(* CODESYS project rsCommSerial.library
   Company: ESO
   Description: Library for Serial communication.
      Depends on rsCommCommon.library
   Version: 0.2.0.3
   Placeholder: ESO LDC Comm Serial Library
   Title: ESO LDC Comm Serial Library

Project tree, tasks and I/O mapping:
  libraries: ESO LDC Comm Common Library, 0.2.0.3 (ESO); Tc2_SerialCom, * (Beckhoff Automation GmbH); Tc2_Standard, * (Beckhoff Automation GmbH); Tc2_System, * (Beckhoff Automation GmbH); Tc2_Utilities, * (Beckhoff Automation GmbH); Tc3_Module, * (Beckhoff Automation GmbH); VisuDialogs, * (System)
  config/
    CCC__1HE_4HE__CoE.jpg
    EL6002_Lakeshore340.xti
    ic0fbiCCC_TwinCAT.fbmap
    LS218_CoE.jpg
    LS340_CoE.jpg
  00000000-0000-0000-0000-000000000000|config\CCC__1HE_4HE__CoE.jpg
  00000000-0000-0000-0000-000000000000|config\EL6002_Lakeshore340.xti
  00000000-0000-0000-0000-000000000000|config\ic0fbiCCC_TwinCAT.fbmap
  00000000-0000-0000-0000-000000000000|config\LS218_CoE.jpg
  00000000-0000-0000-0000-000000000000|config\LS340_CoE.jpg
  DUTs/
    Enumerated/
      Comm/
        data type E_MODBUS_CMD
        data type E_MODBUS_ERROR
        data type E_MODBUS_STATE
        data type E_MODBUS_STATUS
      Devices/
        data type E_CCC_ERROR
        data type E_CCC_STATUS
        data type E_JUMO_ADDRESS
    Structures/
      Comm/
        data type T_MODBUS_CFG
        data type T_MODBUS_CTRL
        data type T_MODBUS_INFO
        data type T_MODBUS_STAT
        data type T_USB_COMM_CFG
      Devices/
        data type T_CCC_CFG
        data type T_CCC_COMMAND
        data type T_CCC_CTRL
        data type T_CCC_INFO
        data type T_CCC_READING
        data type T_CCC_STAT
        data type T_JUMO_CFG
        data type T_JUMO_CTRL
        data type T_JUMO_INFO
        data type T_JUMO_STAT
  GVLs/
  lib/
  POUs/
    Comm/
      function block FB_MODBUS_COMM_BASE [ST]: M_ActionInitExecute, M_ActivityConnect, M_ComPortControl, M_CRC, M_GetHighByte, M_GetINT, M_GetLowByte, M_Reset
      function block FB_MODBUS_COMM_JUMO [ST]
      function block FB_MODBUS_COMM_NO_SIM [ST]
      function block FB_RS_COMM_BASE [ST]: M_ActionInitExecute, M_ActivityConnect, M_ComPortControl, M_GetInitialised, M_GetStatus, M_Reset
      function block FB_RS_COMM_LAKESHORE [ST]: M_ActionInitExecute, M_ComPortControl, M_Reset
      function block FB_RS_COMM_NO_SIM [ST]: M_ActionInitExecute, M_ComPortControl, M_Reset
      function block FB_USB_COMM_NO_SIM [ST]: M_ActionInitExecute, M_ActivityConnect, M_ComPortControl
    Devices/
      function block FB_CCC [ST]: ActivityInitializing, ActivityMonitoring, M_ConvertTemp, M_SetAllFaulty, M_TrimDevReply, M_UpdateDevFlows, M_UpdateDevStatus, M_UpdateDevTemps
      function block FB_JUMO [ST]: ActivityInitializing, ActivityMonitoring, M_ByteSwapFLOAT, M_ByteSwapINT, M_ExtractReadings, M_GetFirstSlaveIndex, M_GetNextSlaveIndex, M_SetCommand, M_UserConfigure
      function block FB_LAKESHORE_RS [ST]: M_Configure, M_GetCommInitialised, M_GetCommStatus, M_GetCouplerState, M_UpdateStatus
    program MAIN [ST]
  VISUs/
    Templates/
      visualisation GUI_TEMPLATE_CCC
      visualisation GUI_TEMPLATE_LAKESHORE_340
      visualisation GUI_TEMPLATE_USB_COMM
    visualisation GUI_ADS_COMM_TEST
    visualisation GUI_CCC
    visualisation GUI_LAKESHORE_340
  text list GlobalTextList
*)

// DUTs/Enumerated/Comm/E_MODBUS_CMD
{attribute 'qualified_only'}
////{xxxattribute 'strict'}
TYPE E_MODBUS_CMD :
(
	NONE		:=	0,
	INIT		:=	1,
	SEND		:=	2
);
END_TYPE

// DUTs/Enumerated/Comm/E_MODBUS_ERROR
{attribute 'qualified_only'}
//{xxxattribute 'strict'}
TYPE E_MODBUS_ERROR :
(
	OK					:= 0,
	NOT_IN_OP_STATE,
	NOT_INIT,
	TIMEOUT,
	SEND,
	RECEIVE,
	WRONG_STATE,
	NOT_IDLE
);
END_TYPE

// DUTs/Enumerated/Comm/E_MODBUS_STATE
{attribute 'qualified_only'}
{attribute 'strict'}
TYPE E_MODBUS_STATE :
(
	NOT_INIT			:= 0,
	IDLE				:= 1,
	RESET				:= 3,
	PREPARE_SEND		:= 5,
	SEND				:= 10,
	RECEIVE				:= 15,
	CLEAR_BUFFER		:= 40,

	ERROR				:= 100
);
END_TYPE

// DUTs/Enumerated/Comm/E_MODBUS_STATUS
{attribute 'qualified_only'}
////{xxxattribute 'strict'}
TYPE E_MODBUS_STATUS :
(
	NOT_INIT	:= -1,
	IDLE		:= 0,
	BUSY		:= 1,
	ERROR		:= 2
);
END_TYPE

// DUTs/Enumerated/Devices/E_CCC_ERROR
TYPE E_CCC_ERROR :
(
	OK				:= 16#0000,
	NOT_IN_OP_STATE	:= 16#0001,
	NOT_INIT		:= 16#0002,
	TIMEOUT			:= 16#0004,
	COMM			:= 16#0008,
	WRONG_STATE		:= 16#0010,
	NOT_IDLE		:= 16#0020
);
END_TYPE

// DUTs/Enumerated/Devices/E_CCC_STATUS
TYPE E_CCC_STATUS :
(
	NOT_INIT	:= -1,
	IDLE		:= 0,
	ERROR		:= 1,
	BUSY		:= 2
);
END_TYPE

// DUTs/Enumerated/Devices/E_JUMO_ADDRESS
TYPE E_JUMO_ADDRESS :
(
	COMMON		:=	0,
	SET_POINTS,
	END
);
END_TYPE

// DUTs/Structures/Comm/T_MODBUS_CFG
TYPE T_MODBUS_CFG EXTENDS T_RS_COMM_CFG:
STRUCT
END_STRUCT
END_TYPE

// DUTs/Structures/Comm/T_MODBUS_CTRL
TYPE T_MODBUS_CTRL :
STRUCT
	nCommand:	E_MODBUS_CMD 	:= E_MODBUS_CMD.NONE;			// Command Number, e.g. to INIT or SEND a command
	bExecute:	BOOL;								// Setting to TRUE activates command
	nSlaveID:	BYTE 	:= 1;						// Modbus Slave ID, 1..247
	nCmdType:	E_MODBUS_CMD_TYPE	:= E_MODBUS_CMD_TYPE.READ;	// Command type; 0-Read, 1-Write
	nRegister:	DINT;								// Command register
	nWords:		DINT	:= 1;						// Number of words
	nValue:		DINT;								// Parameter value

END_STRUCT
END_TYPE

// DUTs/Structures/Comm/T_MODBUS_INFO
TYPE T_MODBUS_INFO :
STRUCT
(*
	Driver Information

	Change LOG:
	01/09/2016:	0.1	- First version. Based on FB_RS_COMM.
	05/09/2016:	0.2	- Implemented Modbus protocol.
	09/11/2016:	0.3	- Status cleared on INIT.
*)

	sDate:			STRING(32)	:= '2016-11-09';
	sDescription:	STRING(80) 	:= 'IR-301 Black Body RS-232 Modbus Driver';
	sName:			STRING(64)	:= 'FB_RS_COMM';
	sPlatform:		STRING(32)	:= 'CoDeSys';
	sSynopsis:		STRING(64)	:= 'IR-301 Black Body RS-232 Modbus Driver';
	nVersionMajor:	DINT		:= 0;
	nVersionMinor:	DINT		:= 3;


END_STRUCT
END_TYPE

// DUTs/Structures/Comm/T_MODBUS_STAT
TYPE T_MODBUS_STAT EXTENDS T_RS_COMM_STAT:
STRUCT
	DeviceReply: 		ARRAY [0..300] OF BYTE;
	nValue:				DINT;	// Value read from the device
END_STRUCT
END_TYPE

// DUTs/Structures/Comm/T_USB_COMM_CFG
TYPE T_USB_COMM_CFG EXTENDS T_RS_COMM_CFG:
STRUCT
	ComPort: 		UDINT :=5;         					// Serial port number [1..255]
    Baudrate: 		UDINT :=57600;						// Baudrate
    Parity: 		ComParity_t :=ComParity_t.PARITY_NONE;			// PARITY_NONE, _EVEN, _ODD, _MARK or _SPACE
    DataBits: 		INT :=8;           					// Data Bits [4..8]
    StopBits: 		ComStopBits_t :=ComStopBits_t.STOPBITS_ONE;		// Stop Bits

    DTR: 			ComDTRCtrl_t :=ComDTRCtrl_t.DTR_CTRL_DISABLE; 	// DTR_CTRL_DISABLE, _ENABLE or _HANDSHAKE
    RTS: 			ComRTSCtrl_t :=ComRTSCtrl_t.RTS_CTRL_DISABLE; 	// RTS_CTRL_DISABLE, _ENABLE, _HANDSHAKE or _TOGGLE
    CTS: 			BOOL :=FALSE;      					// 'Clear to Send' signal
    DSR: 			BOOL :=FALSE;      					// 'Dataset Ready' signal

END_STRUCT
END_TYPE

// DUTs/Structures/Devices/T_CCC_CFG
TYPE T_CCC_CFG EXTENDS T_RS_BASE_CFG:
STRUCT
	CCC_CMD_GET_VERS:	STRING(8) := '>00V??';
	CCC_CMD_RESET:		STRING(8) := '>00u??';
	CCC_CMD_GET_TEMP:	STRING(8) := '>00H??';
	CCC_CMD_GET_FLOW:	STRING(8) := '>00f??';
	CCC_CMD_GET_STAT:	STRING(8) := '>00o??';
	CCC_CMD_SET_HOST:	STRING(8) := '>00J??';
	CCC_CMD_SET_THST:	STRING(8) := '>00T??';
	CCC_CMD_SET_TAMB:	STRING(8) := '>00t??';

	(* List of INIT commands *)
	cmdList_Init:	ARRAY [1..4] OF T_CCC_COMMAND := [
							(cmd := CCC_CMD_RESET, 		nValues := 0),
							(cmd := CCC_CMD_GET_VERS, 	nValues := 0),
							(cmd := '', 				nValues := 0),
							(cmd := '', 				nValues := 0)];


	(*	List of READ commands *)
	cmdList_Read:	ARRAY [1..4] OF T_CCC_COMMAND := [
							(cmd := CCC_CMD_GET_STAT, 	nValues := 5), (* 5 bytes *)
							(cmd := CCC_CMD_GET_TEMP, 	nValues := 5), (* 5 words = 10 bytes*)
							(cmd := CCC_CMD_GET_FLOW, 	nValues := 3), (* 3 words = 6 bytes *)
							(cmd := '', 				nValues := 0)];

END_STRUCT
END_TYPE

// DUTs/Structures/Devices/T_CCC_COMMAND
TYPE T_CCC_COMMAND :
STRUCT
	cmd:		STRING(8);	(* Command to send *)
	nValues:	DINT;   	(* Number of returned numbers (values) in the reply *)
END_STRUCT
END_TYPE

// DUTs/Structures/Devices/T_CCC_CTRL
TYPE T_CCC_CTRL  EXTENDS T_RS_BASE_CTRL:
STRUCT
	(* CTRL *)
END_STRUCT
END_TYPE

// DUTs/Structures/Devices/T_CCC_INFO
TYPE T_CCC_INFO :
STRUCT
(*
	Driver Information

	Change LOG:
	1.0	12/02/2014	- Ported from TC2.
	1.1	13/02/2014	- Addition of input parameters for Model and readout period.
	1.2	20/02/2014	- E_CCC_STATUS.ERROR := 1, to match IODev ICD.
					- Disabled OPC UA for comm instance of FB_RS_COMM.
					- Fixed bug in INIT (wrong pointer used)
					- Bytes swapped for Temperatures and Flows.
					- On error, all values set to 9999. Alarm activated.
	1.3 07/11/2014	- Newest version always for References.
					- Remove Tc2_OpcUa library from References.
					- Renamed library to CCC.library (was CCC_TC3.library)
					- Created lib directory.
	1.4 10/02/2016	- On reboot, the device is in NOT INIT (no error!)
					- On INIT start, error is cleared.
	2.0 2016-08-10	- OPC UA notation with TMC Files
	2.1 2017-02-03	- sCmdSuffix and sReplySuffix passed to comm instance.

*)
	sDate:			STRING(16)	:= '2017-02-03';
	sDescription:	STRING(32) 	:= 'Cabinet Cooling Controller';
	sName:			STRING(16)	:= 'FB_CCC';
	sPlatform:		STRING(16)	:= 'CoDeSys';
	sSynopsis:		STRING(48)	:= 'Cabinet Cooling Controller for models 1HE & 4HE';
	nVersionMajor:	DINT		:= 2;
	nVersionMinor:	DINT		:= 1;

END_STRUCT
END_TYPE

// DUTs/Structures/Devices/T_CCC_READING
TYPE T_CCC_READING :
STRUCT
	Value:	LREAL;
END_STRUCT
END_TYPE

// DUTs/Structures/Devices/T_CCC_STAT
TYPE T_CCC_STAT EXTENDS T_RS_BASE_STAT:
STRUCT
	(* STAT *)
	nRetries:			INT := 0;			// Total number of retries in case of communication problems
	
	bPeriodic:			BOOL := FALSE;		(* Flag if device is reading periodically *)

	sReply:				STRING; 			(* Last Reply to predefined commands*)
	
	sDeviceID:			STRING(48);
	
	(* Status retrieved with command CCC_CMD_GET_STAT *)
	(* decode CSTAT1 byte *)
	bWarn_cabinet_high:			BOOL;
	bWarn_cabinet_no_control:	BOOL;
	bWarn_outlet_high:			BOOL;
	bWarn_inlet_high:			BOOL;
	bWarn_airflow_insufficient:	BOOL;
	bWarn_coolant_insufficient:	BOOL;
	bWarn_door_open:			BOOL;
	bWarn_relay1_warning:		BOOL;
	bWarn_relay2_alarm:			BOOL;

	(* decode CSTAT2 byte *)
	bFault_temp_sensor_ambient:	BOOL;
	bFault_temp_sensor_cabinet:	BOOL;
	bFault_temp_sensor_inlet:	BOOL;
	bFault_temp_sensor_outlet:	BOOL;
	bFault_analog_supply:		BOOL;
	bFault_digital_supply:		BOOL;
	
	(* Temperatures [degC] retrieved with command CCC_CMD_GET_TEMP *)
	lrTemp_outlet:	LREAL;
	lrTemp_inlet:	LREAL;
	lrTemp_cabinet:	LREAL;
	lrTemp_ambient:	LREAL;
	
	(* Flows [l/h] retrieved with command CCC_CMD_GET_FLOW *)
	lrFlow_1:		LREAL;
	lrFlow_2:		LREAL;
	lrFlow_3:		LREAL;

END_STRUCT
END_TYPE

// DUTs/Structures/Devices/T_JUMO_CFG
TYPE T_JUMO_CFG EXTENDS T_RS_BASE_CFG:
STRUCT
	// Register Addresses
	nAddrCommon:		INT	:= 16#00A4;
	nAddrSetPoints:		INT	:= 16#083C;

	// Number of bytes to read
	// These are ONLY data bytes. Total bytes to read is higher (+5) 
	nWordsCommon:		INT	:= 116;	// 232 bytes
	nWordsSetPoints:	INT	:= 32;	// 32 words
	
	aSlaveID:			ARRAY [1..8] OF BYTE := [1,2,3,4,5,6,7,8];
	aDevUsed:			ARRAY [1..8] OF BOOL := [TRUE, 7(FALSE)];	// Only first JUMO used by default
	
END_STRUCT
END_TYPE

// DUTs/Structures/Devices/T_JUMO_CTRL
TYPE T_JUMO_CTRL EXTENDS T_RS_BASE_CTRL:
STRUCT
	nSlaveID:	BYTE 	:= 1;						// Modbus Slave ID, 1..247
	nCmdType:	DINT	:= E_MODBUS_CMD_TYPE.READ;	// Command type; 0-Read, 1-Write
	nRegister:	DINT;								// Command register
	nWords:		DINT	:= 1;						// Number of words
	nValue:		DINT;								// Parameter value
END_STRUCT
END_TYPE

// DUTs/Structures/Devices/T_JUMO_INFO
TYPE T_JUMO_INFO :
STRUCT
(*
	Driver Information

	Change LOG:
	1.0	12/02/2014	- Copied from VLT.
*)
	sDate:			STRING(16)	:= '2016-08-10';
	sDescription:	STRING(32) 	:= 'JUMO controller';
	sName:			STRING(16)	:= 'FB_JUMO';
	sPlatform:		STRING(16)	:= 'CoDeSys';
	sSynopsis:		STRING(48)	:= 'EtherCAT PLC JUMO controller';
	nVersionMajor:	DINT		:= 1;
	nVersionMinor:	DINT		:= 0;

END_STRUCT
END_TYPE

// DUTs/Structures/Devices/T_JUMO_STAT
TYPE T_JUMO_STAT EXTENDS T_RS_BASE_STAT:
STRUCT

	nRetries:				INT := 0;	// Total number of retries in case of communication problems
	
	nInputBuffer: 			ARRAY [0..300] OF BYTE;	// Binary data read from JUMO

	// Data for up to 8 JUMO devices (4 TeePee units) daisy chained
	// Data for the first 4 control loops [1-4]
	// ARRAY[<device>,<control loop>, <value>]
	aSetPoints:				ARRAY [1..8,1..4,1..4] OF REAL;
	aCtrlParams:			ARRAY [1..8,1..4,1..9] OF REAL;
	aSwitchStats:			ARRAY [1..8,1..4,1..2] OF INT;

	// 8 analog inputs per JUMO
	aAnalogInputs:			ARRAY [1..8,1..8] OF REAL;
	aMath:					ARRAY [1..8,1..8] OF REAL;

	aSamplingTime:			ARRAY [1..8] OF REAL;
	aInternalTemperature:	ARRAY [1..8] OF REAL;
END_STRUCT
END_TYPE

// POUs/Comm/FB_MODBUS_COMM_BASE
FUNCTION_BLOCK FB_MODBUS_COMM_BASE
VAR_INPUT
	in_bSimulation:		BOOL := FALSE;
	in_nModel:			DINT;	// Device model number. Zero if N/A.
	in_cReadFunction:	BYTE := 3;	// Function used for READ. MUST be 3 or 4.
END_VAR
VAR_OUTPUT
END_VAR
VAR CONSTANT
END_VAR
VAR
	{attribute 'OPC.UA.DA' := '1'}
	cfg:		T_MODBUS_CFG;				// Config parameters
	{attribute 'OPC.UA.DA' := '1'}
	ctrl:		T_MODBUS_CTRL;				// Control parameters
	{attribute 'OPC.UA.DA' := '1'}
	{attribute 'OPC.UA.DA.Access' := '1'}
	info:		T_MODBUS_INFO; 				// Info parameters - ReadOnly
	{attribute 'OPC.UA.DA' := '1'}
	{attribute 'OPC.UA.DA.Access' := '1'}
	stat:		T_MODBUS_STAT;				// Status parameters - ReadOnly

	{attribute 'OPC.UA.DA' := '0'}
	simRef:		REFERENCE TO FB_SIM_MODBUS_COMM_BASE;	// Reference to COMM simulator


	(***** Physical signals - to be mapped to EL60xx serial port terminal !!! *****)
	COMin_EL60xx	AT %I* 	: KL6inData22B;	(* linked to the EL60xx *)
	COMout_EL60xx	AT %Q*	: KL6outData22B;(* linked to the EL60xx *)
	i_nCouplerState	AT %I*	: UINT;			(* Link it to Coupler->InfoData->State *)

	(* Serial line control *)
	COMportControl: 		SerialLineControl;
	RxBuffer:				ComBuffer;		(* Receive data buffer; used with all receive function blocks *)
	TxBuffer:				ComBuffer;		(* Transmit data buffer; used with all receive function blocks *)


	(* Send/Receive FB's and VAR's *)
	Receive: 			ReceiveData;
	Send:				SendData;
	ClearComBufferTx:	ClearComBuffer;
	ClearComBufferRx:	ClearComBuffer;
	ComReset:			ComReset;

	(* Timers *)
	fbTimer:			TON; (* Timeout for RECEIVE *)

	State:				INT := E_MODBUS_STATE.NOT_INIT;
	nextState:			INT := E_MODBUS_STATE.IDLE;


	cmd:				STRING(16);		// Only first 8 bytes are used

	nBytesToReceive:	UDINT;			// 8 for command, 7 for status
	nBytesToSend:		UDINT := 8;		// Always 8

	crc:				WORD;			// CRC Check word

	i:					INT;
END_VAR

(* ============================================
	Check if the HW is OK. 
	The coupler state must be 8, i.e. OPERATIONAL.
============================================== *)
IF i_nCouplerState <> 8  AND  NOT in_bSimulation THEN	(* If the hardware status is NOT OK, we cannot trust the readings. *)
	stat.nErrorCode	:= M_GetINT(E_MODBUS_ERROR.NOT_IN_OP_STATE);
	stat.sErrorText	:= 'Not in OPERATIONAL state. Check if variable i_nCouplerState is linked to HW.';
	stat.nStatus	:= M_GetINT(E_MODBUS_STATUS.ERROR);
	stat.sStatus	:= 'ERROR';
	RETURN;
END_IF


//
// Execute Simulator, if in simulation
//
IF in_bSimulation  THEN
	simRef(in_nModel := in_nModel);
END_IF


(*====================================================
	Handling of commands sent through OPC UA interface.
	Executed only when flag bExecute goes from LOW to HIGH.
	bExecute is reset by the PLC application.
=====================================================*)

IF ctrl.bExecute THEN
	ctrl.bExecute	:= FALSE;
	(* Save last command and reset the command *)
	stat.nLastCommand 	:= M_GetINT(ctrl.nCommand);
	ctrl.nCommand		:= E_MODBUS_CMD.NONE;

	(* Commands can only be sent when device is IDLE *)
	IF INT_TO_DINT(stat.nLastCommand) <> INT_TO_DINT(E_MODBUS_CMD.INIT)  AND  State <> E_MODBUS_STATE.IDLE THEN
		State 			:= E_MODBUS_STATE.ERROR;
		stat.nStatus	:= M_GetINT(E_MODBUS_STATUS.ERROR);
		stat.sStatus	:= 'ERROR';
		stat.nErrorCode	:= M_GetINT(E_MODBUS_ERROR.NOT_IDLE);
		stat.sErrorText	:= 'Device busy. Should be in IDLE to receive commands.';
		RETURN;
	END_IF


	(* Device has to be initialised before being used *)
	IF INT_TO_DINT(stat.nLastCommand) <> INT_TO_DINT(E_MODBUS_CMD.INIT) THEN
		IF NOT stat.bInitialised  THEN
			State 			:= E_MODBUS_STATE.ERROR;
			stat.nStatus	:= M_GetINT(E_MODBUS_STATUS.ERROR);
			stat.sStatus	:= 'ERROR';
			stat.nErrorCode	:= M_GetINT(E_MODBUS_ERROR.NOT_INIT);
			stat.sErrorText	:= 'Device not initialised.';
			RETURN;
		END_IF
	END_IF



	CASE stat.nLastCommand OF
	E_RS_COMM_CMD.INIT:
		// Comm port specific.
		// M_ActionInitExecute() has to set next State!!!
		M_ActionInitExecute();

	E_RS_COMM_CMD.SEND:
		stat.nErrorCode	:= M_GetINT(E_MODBUS_ERROR.OK);
		stat.nStatus	:= M_GetINT(E_MODBUS_STATUS.BUSY);
		stat.sErrorText	:= 'OK';
		stat.sStatus	:= 'BUSY';
		State 			:= E_MODBUS_STATE.PREPARE_SEND;

	END_CASE

END_IF



(*====================================================
	Background communication with KL60xx terminal.
	Called only during Send or Receive!!!
	It communicates with the serial line hardware device and 
	transmits or receives data.
=====================================================*)

CASE State OF
E_MODBUS_STATE.IDLE,
E_MODBUS_STATE.CLEAR_BUFFER,
E_MODBUS_STATE.SEND,
E_MODBUS_STATE.RECEIVE:

	COMportControl(
		Mode		:= ComSerialLineMode_t.SERIALLINEMODE_KL6_22B_STANDARD,
		pComIn		:= ADR(COMin_EL60xx),				(* I/O data; see global variables *)
		pComOut		:= ADR(COMout_EL60xx),				(* I/O data; see global variables *)
		SizeComIn	:= UINT_TO_INT(SIZEOF(COMin_EL60xx)),			(* I/O data; see global variables *)
		TxBuffer	:= TxBuffer,						(* transmit buffer; see global variables *)
		RxBuffer	:= RxBuffer);						(* receive buffer; see global variables *)

END_CASE





(*======================
=======================
 	State machine 
=======================
=======================*)

CASE State OF

E_MODBUS_STATE.ERROR:
	ClearComBufferTx (Buffer := TxBuffer);
	ClearComBufferRx (Buffer := RxBuffer);
	stat.nStatus	:= M_GetINT(E_MODBUS_STATUS.ERROR);
	stat.sStatus	:= 'ERROR';
	State 			:= E_MODBUS_STATE.IDLE;
	RETURN;


E_MODBUS_STATE.NOT_INIT:
	ClearComBufferTx (Buffer := TxBuffer);
	ClearComBufferRx (Buffer := RxBuffer);
	stat.bInitialised	:= FALSE;
	stat.nErrorCode		:= M_GetINT(E_MODBUS_ERROR.OK);
	stat.sErrorText		:= 'OK';
	stat.nStatus		:= M_GetINT(E_MODBUS_STATUS.NOT_INIT);
	stat.sStatus		:= 'NOT INIT';


E_MODBUS_STATE.IDLE:
	(* Nothing to do in IDLE *)
	RETURN;


E_MODBUS_STATE.RESET:
	(* Reset the connected serial hardware *)
	ComReset (
		Execute 	:= TRUE,
		pComIn		:= ADR(COMin_EL60xx),
		pComOut		:= ADR(COMout_EL60xx),
		SizeComIn	:= SIZEOF(COMin_EL60xx),
		);

	(* Next step is to clear the buffers *)
	IF ComReset.Done THEN
		fbTimer (IN := FALSE);	// Reset the timer
		State 		:= E_MODBUS_STATE.CLEAR_BUFFER;
	END_IF
	RETURN;


E_MODBUS_STATE.PREPARE_SEND:
	(*******************************************************************************************
	Here we set the command string, i.e. add suffix if not included in the command.
	Then, the state is changed to  E_MODBUS_STATE.SEND.
	********************************************************************************************)

	(* Clear reply string *)
	MEMSET(ADR(stat.DeviceReply), 0 , SIZEOF(stat.DeviceReply) );

	cmd	:= '';
	cmd[0] := ctrl.nSlaveID;
	cmd[2] := M_GetHighByte(ctrl.nRegister);
	cmd[3] := M_GetLowByte(ctrl.nRegister);
	IF ctrl.nCmdType = E_MODBUS_CMD_TYPE.WRITE  THEN
		cmd[1] := 6;			// Write Function
		nBytesToReceive	:= 8;	// Reply equals Command
		cmd[4] := M_GetHighByte(ctrl.nValue);
		cmd[5] := M_GetLowByte(ctrl.nValue);
	ELSE
		cmd[1] := in_cReadFunction;			// Read Function (3 or 4)
		nBytesToReceive	:= DINT_TO_UDINT(2 * ctrl.nWords  +  5); 
		// Bytes 4..5, receive one word (2 bytes)
		cmd[4] := M_GetHighByte(ctrl.nWords);
		cmd[5] := M_GetLowByte(ctrl.nWords);
	END_IF
	
	// Calculate CRC for the first 6 bytes
	crc	:= M_CRC(ADR(cmd),6);
	
	cmd[6] := M_GetLowByte(crc);
	cmd[7] := M_GetHighByte(crc);
	
	IF in_bSimulation THEN
		fbTimer (IN := FALSE); 	(* reset timer *)
		ClearComBufferRx (Buffer := RxBuffer);
		stat.sReply		:= simRef.M_GetSimReply(cmd);	// Get simulated reply
		FOR i:=0 TO 255 DO
			stat.DeviceReply[i] := stat.sReply[i];
		END_FOR
		stat.nStatus	:= M_GetINT(E_MODBUS_STATUS.IDLE);
		stat.sStatus	:= 'IDLE';
		State 			:= E_MODBUS_STATE.IDLE;
	ELSE	
		ClearComBufferTx (Buffer := TxBuffer);
		stat.nStatus	:= M_GetINT(E_MODBUS_STATUS.BUSY);
		stat.sStatus	:= 'BUSY';
		State 			:= E_MODBUS_STATE.SEND;
	END_IF
	RETURN;


E_MODBUS_STATE.SEND:

	(* Send the command via serial port. *)
	Send(
		pSendData	:= ADR(cmd),
		Length		:= nBytesToSend,
		TXbuffer	:= TxBuffer);

	(* If the string was not sent in one cycle, go to next cycle *)
	IF Send.Busy THEN
		RETURN;
	ELSE
		IF Send.Error <> ComError_t.COMERROR_NOERROR THEN
			State 			:= E_MODBUS_STATE.ERROR;
			stat.nErrorCode	:= M_GetINT(E_MODBUS_ERROR.SEND);
			stat.sErrorText	:= 'Send Failed';
		ELSE
			fbTimer (IN := FALSE);	// reset timer
			// One extra call of background communication
			COMportControl(
				Mode		:= ComSerialLineMode_t.SERIALLINEMODE_KL6_22B_STANDARD,
				pComIn		:= ADR(COMin_EL60xx),				(* I/O data; see global variables *)
				pComOut		:= ADR(COMout_EL60xx),				(* I/O data; see global variables *)
				SizeComIn	:= UINT_TO_INT(SIZEOF(COMin_EL60xx)),			(* I/O data; see global variables *)
				TxBuffer	:= TxBuffer,						(* transmit buffer; see global variables *)
				RxBuffer	:= RxBuffer);						(* receive buffer; see global variables *)

			State := E_MODBUS_STATE.RECEIVE; 	(* Next state is RECEIVE *)
		END_IF
		RETURN;
	END_IF



E_MODBUS_STATE.RECEIVE:
	(* Start the 3 sec timeout timer for receive *)
	fbTimer (IN := TRUE, PT := T#3S);

	(* Check for timeout. Goto ERROR if timeout expired. *)
	IF fbTimer.Q THEN
		fbTimer (IN := FALSE); (* reset timer *)

		State 			:= E_MODBUS_STATE.ERROR;
		stat.nErrorCode	:= M_GetINT(E_MODBUS_ERROR.TIMEOUT);
		stat.sErrorText	:= 'Timeout on Receive';
		RETURN;
	END_IF

	// Wait for the reply.
	// Terminate read 1000 ms after receiving the first character.
	Receive(
		pReceiveData	:= ADR(stat.DeviceReply),
		SizeReceiveData := nBytesToReceive,
		Timeout			:= T#1000MS,
		Reset			:= FALSE,
		RXbuffer		:= RxBuffer);


	(* Check for possible errors *)
	IF Receive.Error <> ComError_t.COMERROR_NOERROR THEN
		fbTimer (IN := FALSE);	(* reset timer *)

		State 			:= E_MODBUS_STATE.ERROR;
		stat.nErrorCode	:= M_GetINT(E_MODBUS_ERROR.RECEIVE);
		stat.sErrorText	:= 'Receive Failed';
		RETURN;
	END_IF

	(* Handle reply *)
	IF Receive.DataReceived THEN
		(* We have received a reply. Reset timers and triggers. *)
		fbTimer (IN := FALSE); 	(* reset timer *)

		// Calculate CRC for the first (nBytesToReceive-2) bytes.
		// The last two bytes are the CRC returned by the device.
		// Do a CRC check.
		crc	:= M_CRC(ADR(stat.DeviceReply),UDINT_TO_INT(nBytesToReceive-2));
		
		IF stat.DeviceReply[nBytesToReceive-1] <> M_GetHighByte(crc) THEN
			State 			:= E_MODBUS_STATE.ERROR;
			stat.nErrorCode	:= M_GetINT(E_MODBUS_ERROR.RECEIVE);
			stat.sErrorText	:= 'Received CRC does not match';
			RETURN;
		ELSIF stat.DeviceReply[nBytesToReceive-2] <> M_GetLowByte(crc) THEN
			State 			:= E_MODBUS_STATE.ERROR;
			stat.nErrorCode	:= M_GetINT(E_MODBUS_ERROR.RECEIVE);
			stat.sErrorText	:= 'Received CRC does not match';
			RETURN;
		END_IF
	
		
		(* Clear the receive buffer ONLY when all replies have been received! *)
		ClearComBufferRx (Buffer := RxBuffer);
		State 			:= E_MODBUS_STATE.IDLE;
		stat.nStatus	:= M_GetINT(E_MODBUS_STATUS.IDLE);
		stat.sStatus	:= 'IDLE';
		RETURN;
	ELSIF Receive.RxTimeout THEN
		(* Handle reply *)
		(* We have received a reply. Reset timers and triggers. *)
		fbTimer (IN := FALSE); 	(* reset timer *)

		// Clear the receive buffer
		ClearComBufferRx (Buffer := RxBuffer);

		stat.nErrorCode	:= M_GetINT(E_MODBUS_ERROR.TIMEOUT);
		stat.sErrorText	:= 'Did not receive expected number of bytes';

		State 			:= E_MODBUS_STATE.ERROR;
		RETURN;
	END_IF



E_MODBUS_STATE.CLEAR_BUFFER:
	// Read all characters present in the receive buffer.
	// Keep reading for 1 sec.
	fbTimer (IN := TRUE, PT := T#1S);
	IF fbTimer.Q THEN
		(* reset timer *)
		fbTimer (IN := FALSE);
		stat.bInitialised	:= TRUE;
		stat.nStatus		:= M_GetINT(E_MODBUS_STATUS.IDLE);
		stat.sStatus		:= 'INITIALISED';
		State 				:= E_MODBUS_STATE.IDLE;
		RETURN;
	END_IF

	Receive(
		pReceiveData	:= ADR(stat.DeviceReply),
		SizeReceiveData := SIZEOF(nBytesToReceive),
		Timeout			:= T#300MS,
		Reset			:= FALSE,
		RXbuffer		:= RxBuffer);



ELSE
(* Unsuported state *)
	State 			:= E_MODBUS_STATE.ERROR;
	stat.nErrorCode	:= M_GetINT(E_MODBUS_ERROR.WRONG_STATE);
	stat.sErrorText	:= 'Unknown State';
END_CASE

METHOD M_ActionInitExecute
VAR_INPUT
END_VAR
//
// If in simulation, there is no need to reset anything.
// Just set it to initialised and go to IDLE state.
//
IF in_bSimulation THEN
	fbTimer (IN := FALSE);	// Reset timer
	stat.bInitialised	:= TRUE;
	stat.nStatus		:= M_GetINT(E_MODBUS_STATUS.IDLE);
	stat.sStatus		:= 'INITIALISED';
	State 				:= E_MODBUS_STATE.IDLE;
ELSE
	stat.bInitialised	:= FALSE;
	stat.sStatus		:= 'INITIALISING';
	stat.nStatus		:= M_GetINT(E_MODBUS_STATUS.BUSY);
	stat.nErrorCode		:= M_GetINT(E_MODBUS_ERROR.OK);
	stat.sErrorText		:= 'OK';

	// Reset the connected serial hardware 
	ComReset (
		Execute 	:= FALSE,
		pComIn		:= ADR(COMin_EL60xx),
		pComOut		:= ADR(COMout_EL60xx),
		SizeComIn	:= SIZEOF(COMin_EL60xx),
		);

	// Set next state
	State 	:= E_MODBUS_STATE.RESET;
END_IF
END_METHOD

METHOD M_ActivityConnect
VAR_INPUT
END_VAR
// TODO: Implement in extended FB
END_METHOD

METHOD M_ComPortControl
VAR_INPUT
END_VAR
// TODO: Implement in extended FB
END_METHOD

METHOD M_CRC : WORD
VAR_INPUT
	p:	POINTER TO BYTE;
	n:	INT;
END_VAR
VAR
  crc: 			WORD;
  bit_count: 	BYTE;
  char_ptr: 	POINTER TO BYTE;
  pos:			INT := 0;
END_VAR
VAR CONSTANT
	POLYNOMIAL: WORD := 16#A001;
END_VAR

// Start at the beginning of the packet
char_ptr := p;

// Initialize CRC
crc := 16#FFFF;

// Loop through the entire packet
WHILE pos < n DO
	
	  // Exclusive-OR the byte with the CRC
	crc := crc XOR char_ptr^;		// crc ^= (unsigned int)*char_ptr;
	
	  // Loop through all 8 data bits
	  bit_count := 0;
	  WHILE bit_count < 8 DO
		  // If the LSB is 1, shift the CRC and XOR
		  // the polynomial mask with the CRC
		  IF (crc AND 16#0001) <> 16#0000 THEN
			
			  crc := SHR(crc,1);	// crc >>= 1;
			  crc := crc XOR POLYNOMIAL;	// crc ^= POLYNOMIAL;
			
		  // If the LSB is 0, shift the CRC only
		  else
			crc := SHR(crc,1);	// crc >>= 1;			
		END_IF
		bit_count := bit_count + 1;
	  END_WHILE
	  char_ptr := char_ptr + 1;
	  pos := pos + 1;
END_WHILE

M_CRC := crc;
END_METHOD

METHOD M_GetHighByte : BYTE
VAR_INPUT
	n:	DINT;
END_VAR
VAR
	w:	WORD;
END_VAR
w := DINT_TO_WORD(n);
M_GetHighByte	:= WORD_TO_BYTE(SHR((w AND 16#FF00), 8));
END_METHOD

METHOD M_GetINT : INT
VAR_INPUT
	nInt:	INT;
END_VAR
M_GetINT	:= nInt;
END_METHOD

METHOD M_GetLowByte : BYTE
VAR_INPUT
	n:	DINT;
END_VAR
VAR
	w:	WORD;
END_VAR
w := DINT_TO_WORD(n);
M_GetLowByte	:= WORD_TO_BYTE((w AND 16#00FF));
END_METHOD

METHOD M_Reset
VAR_INPUT
END_VAR
// TODO: Implement in extended FB
END_METHOD

END_FUNCTION_BLOCK

// POUs/Comm/FB_MODBUS_COMM_JUMO
FUNCTION_BLOCK FB_MODBUS_COMM_JUMO EXTENDS FB_MODBUS_COMM_BASE
VAR_INPUT
END_VAR
VAR_OUTPUT
END_VAR
VAR CONSTANT
END_VAR
VAR
	{attribute 'OPC.UA.DA' := '0'}
	sim:		FB_SIM_MODBUS_COMM_JUMO;	// Reference to COMM simulator

END_VAR

simRef	REF=sim;

// Execute base FB, i.e. FB_MODBUS_COMM_BASE.
SUPER^();

END_FUNCTION_BLOCK

// POUs/Comm/FB_MODBUS_COMM_NO_SIM
FUNCTION_BLOCK FB_MODBUS_COMM_NO_SIM EXTENDS FB_MODBUS_COMM_BASE
VAR_INPUT
END_VAR
VAR_OUTPUT
END_VAR
VAR CONSTANT
END_VAR
VAR
	{attribute 'OPC.UA.DA' := '0'}
	sim:		FB_SIM_MODBUS_COMM_BASE;	// Reference to COMM simulator

END_VAR

simRef	REF=sim;

// Execute base FB, i.e. FB_MODBUS_COMM_BASE.
SUPER^();

END_FUNCTION_BLOCK

// POUs/Comm/FB_RS_COMM_BASE
FUNCTION_BLOCK FB_RS_COMM_BASE
VAR_INPUT
	in_bSimulation:		BOOL := FALSE;
	in_nModel:			DINT;	// Device model number. Zero if N/A.
	in_sCmdSuffix:		STRING(16) := '$0D$0A';	// Terminator for command, default '<CR><LF>'
	in_sReplySuffix:	STRING(16) := '$0D$0A';	// Terminator for reply, default '<CR><LF>'
	in_nTimeout:		DINT := 3000;			// Timeout [ms] on command reply. Default 3000 (3 sec)
END_VAR
VAR_OUTPUT
END_VAR
VAR CONSTANT
END_VAR
VAR
	{attribute 'OPC.UA.DA' := '1'}
	cfgRef:			REFERENCE TO T_RS_COMM_CFG;		// Config parameters
	{attribute 'OPC.UA.DA' := '1'}
	ctrlRef:		REFERENCE TO T_RS_COMM_CTRL;	// Control parameters
	{attribute 'OPC.UA.DA' := '1'}
	{attribute 'OPC.UA.DA.Access' := '1'}
	infoRef:		REFERENCE TO T_RS_COMM_INFO; 	// Info parameters - ReadOnly
	{attribute 'OPC.UA.DA' := '1'}
	{attribute 'OPC.UA.DA.Access' := '1'}
	statRef:		REFERENCE TO T_RS_COMM_STAT;	// Status parameters - ReadOnly

	{attribute 'OPC.UA.DA' := '0'}
	simRef:			REFERENCE TO FB_SIM_RS_COMM_BASE;	// Reference to COMM simulator


	// Physical signals - to be mapped
	i_nCouplerState	AT %I*	: UINT;			(* Link it to Coupler->InfoData->State *)

	(* Serial line control *)
//	COMportControl: 		SerialLineControl;
	RxBuffer:				ComBuffer;		(* Receive data buffer; used with all receive function blocks *)
	TxBuffer:				ComBuffer;		(* Transmit data buffer; used with all receive function blocks *)

	(* Send/Receive FB's and VAR's *)
	Receive: 			ReceiveString255;
	Send:				SendString;
	ClearComBufferTx:	ClearComBuffer;
	ClearComBufferRx:	ClearComBuffer;
	ComReset:			ComReset;

	DeviceReply: 		STRING(255);

	(* Timers *)
	fbTimer:			TON; (* Timeout for RECEIVE *)

	State:				INT := E_RS_COMM_STATE.NOT_INIT;
	nextState:			INT := E_RS_COMM_STATE.IDLE;

	cmd:				STRING;

	nNumReplies:		DINT := 0;

	pos:				INT;
END_VAR

(* ============================================
	Check if the HW is OK. 
	The coupler state must be 8, i.e. OPERATIONAL (if not simulated).
============================================== *)
IF i_nCouplerState <> 8  AND  NOT in_bSimulation  THEN	(* If the hardware status is NOT OK, we cannot trust the readings. *)
	statRef.nErrorCode	:= E_RS_COMM_ERROR.NOT_IN_OP_STATE;
	statRef.sErrorText	:= 'Not in OPERATIONAL state. Check if variable i_nCouplerState is linked to HW.';
	statRef.nStatus		:= E_RS_COMM_STATUS.ERROR;
	statRef.sStatus		:= 'ERROR';
	RETURN;
END_IF

//
// Execute Simulator, if in simulation
//
IF in_bSimulation  THEN
	simRef(in_nModel := in_nModel, in_sReplySuffix := in_sReplySuffix);
END_IF

(*====================================================
	Handling of commands sent through OPC UA interface.
	Executed only when flag bExecute goes from LOW to HIGH.
	bExecute is reset by the PLC application.
=====================================================*)

IF ctrlRef.bExecute THEN
	ctrlRef.bExecute	:= FALSE;
	(* Save last command and reset the command *)
	statRef.nLastCommand 	:= ctrlRef.nCommand;
	ctrlRef.nCommand		:= E_RS_COMM_CMD.NONE;

	(* Commands can only be sent when device is IDLE *)
	IF statRef.nLastCommand <> E_RS_COMM_CMD.INIT  AND  State <> E_RS_COMM_STATE.IDLE THEN
		State 				:= E_RS_COMM_STATE.ERROR;
		statRef.nStatus		:= E_RS_COMM_STATUS.ERROR;
		statRef.sStatus		:= 'ERROR';
		statRef.nErrorCode	:= E_RS_COMM_ERROR.NOT_IDLE;
		statRef.sErrorText	:= 'Device busy. Should be in IDLE to receive commands.';
		RETURN;
	END_IF


	(* Device has to be initialised before being used *)
	IF statRef.nLastCommand <> E_RS_COMM_CMD.INIT THEN
		IF NOT statRef.bInitialised  THEN
			State 				:= E_RS_COMM_STATE.ERROR;
			statRef.nStatus		:= E_RS_COMM_STATUS.ERROR;
			statRef.sStatus		:= 'ERROR';
			statRef.nErrorCode	:= E_RS_COMM_ERROR.NOT_INIT;
			statRef.sErrorText	:= 'Device not initialised.';
			RETURN;
		END_IF
	END_IF



	CASE statRef.nLastCommand OF
	E_RS_COMM_CMD.INIT:
		// Comm port specific.
		// M_ActionInitExecute() has to set next State!!!
		M_ActionInitExecute();

	E_RS_COMM_CMD.SEND:
		statRef.nErrorCode	:= E_RS_COMM_ERROR.OK;
		statRef.nStatus		:= E_RS_COMM_STATUS.BUSY;
		statRef.sErrorText	:= 'OK';
		statRef.sStatus		:= 'BUSY';
		State 				:= E_RS_COMM_STATE.PREPARE_SEND;

	END_CASE

END_IF



(*====================================================
	Background communication with KL60xx terminal.
	Called only during Send or Receive!!!
	It communicates with the serial line hardware device and 
	transmits or receives data.
=====================================================*)

CASE State OF
E_RS_COMM_STATE.IDLE,
E_RS_COMM_STATE.CONNECT,
E_RS_COMM_STATE.CLEAR_BUFFER,
E_RS_COMM_STATE.SEND,
E_RS_COMM_STATE.RECEIVE:
	// Backgroung communication control.
	// This method is just a place holder..
	// TODO: Implement for each communication protocol, i.e. for RS and ADS/USB.
	M_ComPortControl();	

END_CASE





(*======================
=======================
 	State machine 
=======================
=======================*)

CASE State OF

E_RS_COMM_STATE.ERROR:
	ClearComBufferTx (Buffer := TxBuffer);
	ClearComBufferRx (Buffer := RxBuffer);
	statRef.nStatus	:= E_RS_COMM_STATUS.ERROR;
	statRef.sStatus	:= 'ERROR';
	State 			:= E_RS_COMM_STATE.IDLE;
	RETURN;


E_RS_COMM_STATE.NOT_INIT:
	ClearComBufferTx (Buffer := TxBuffer);
	ClearComBufferRx (Buffer := RxBuffer);
	statRef.bInitialised	:= FALSE;
	statRef.nErrorCode		:= E_RS_COMM_ERROR.OK;
	statRef.sErrorText		:= 'OK';
	statRef.nStatus			:= E_RS_COMM_STATUS.NOT_INIT;
	statRef.sStatus			:= 'NOT INIT';


E_RS_COMM_STATE.IDLE:
	(* Nothing to do in IDLE *)
	RETURN;


E_RS_COMM_STATE.CONNECT:
	M_ActivityConnect();

	
E_RS_COMM_STATE.RESET:
	// Specific call of communication reset
	M_Reset();
	RETURN;


E_RS_COMM_STATE.PREPARE_SEND:
	(*******************************************************************************************
	Here we set the command string, i.e. add suffix if not included in the command.
	Then, the state is changed to  E_RS_COMM_STATE.SEND.
	********************************************************************************************)

	(* Clear reply string *)
	DeviceReply	:= '';

	cmd	:= ctrlRef.sCmd;

	statRef.nStatus	:= E_RS_COMM_STATUS.BUSY;
	statRef.sStatus	:= 'BUSY';

	(* Add suffix CR/LF to the user command if missing *)
	pos := FIND(cmd,cfgRef.sCmdSuffix);
	IF pos = 0 THEN
		cmd := CONCAT(cmd, cfgRef.sCmdSuffix);
	END_IF

	//
	// If in simulation, there is no need to send anything.
	// Just get a reply from the simulator and go to IDLE state.
	//
	IF in_bSimulation THEN
		fbTimer (IN := FALSE); 	(* reset timer *)
		ClearComBufferRx (Buffer := RxBuffer);
		statRef.sReply	:= simRef.M_GetSimReply(cmd);	// Get simulated reply
		State 			:= E_RS_COMM_STATE.IDLE;
		statRef.nStatus	:= E_RS_COMM_STATUS.IDLE;
		statRef.sStatus	:= 'IDLE';
	ELSE	
		ClearComBufferTx (Buffer := TxBuffer);
		statRef.nStatus	:= E_RS_COMM_STATUS.BUSY;
		statRef.sStatus	:= 'BUSY';
		nNumReplies		:= 0;		(* Have not received any reply yet. Used for handling multiple replies. *)
		State 			:= E_RS_COMM_STATE.SEND;
	END_IF
	RETURN;


E_RS_COMM_STATE.SEND:
	(* Send the command via serial port. *)
	Send(
		SendString	:= cmd,
		TXbuffer	:= TxBuffer);

	(* If the string was not sent in one cycle, go to next cycle *)
	IF Send.Busy THEN
		RETURN;
	ELSE
		IF Send.Error <> ComError_t.COMERROR_NOERROR THEN
			State 			:= E_RS_COMM_STATE.ERROR;
			statRef.nErrorCode	:= E_RS_COMM_ERROR.SEND;
			statRef.sErrorText	:= 'Send Failed';
		ELSE
			fbTimer (IN := FALSE);	// reset timer
		
			statRef.sReply := ''; 				(* No reply yet *)
		
			(* 	The command has been sent.
				If there is no reply, goto IDLE state.
				Otherwise, goto RECEIVE state. *)
			IF ctrlRef.bHasReply THEN
				State := E_RS_COMM_STATE.RECEIVE; 	(* Next state is RECEIVE *)
			ELSE
				(* Prepare next state *)
				State 			:= E_RS_COMM_STATE.IDLE;	 	(* Next state is IDLE *)
				statRef.nStatus	:= E_RS_COMM_STATUS.IDLE;
				statRef.sStatus	:= 'IDLE';
			END_IF
			RETURN;
		END_IF
	END_IF


E_RS_COMM_STATE.RECEIVE:
	(* Start the timeout timer for receive *)
	fbTimer (IN := TRUE, PT := DINT_TO_TIME(cfgRef.nTimeout+500)); (* 500ms extra timeout for reply *)


	(* Check for timeout. Goto ERROR if timeout expired. *)
	IF fbTimer.Q THEN
		fbTimer (IN := FALSE); (* reset timer *)

		State 			:= E_RS_COMM_STATE.ERROR;
		statRef.nErrorCode	:= E_RS_COMM_ERROR.TIMEOUT;
		statRef.sErrorText	:= 'Timeout on Receive';
		RETURN;
	END_IF

	(* Wait for the reply *)
	Receive(
		Prefix			:= '',
		Suffix			:= cfgRef.sReplySuffix,
		Timeout			:= DINT_TO_TIME(cfgRef.nTimeout),
		ReceivedString	:= DeviceReply,
		RXbuffer		:= RxBuffer,
		Reset			:= FALSE);


	(* Check for possible errors *)
	IF Receive.Error <> ComError_t.COMERROR_NOERROR OR  Receive.RxTimeout THEN
		fbTimer (IN := FALSE);	(* reset timer *)

		State 	:= E_RS_COMM_STATE.ERROR;
		statRef.nErrorCode	:= E_RS_COMM_ERROR.RECEIVE;
		statRef.sErrorText	:= 'Receive Failed';
		RETURN;
	END_IF

	(* Handle reply *)
	IF Receive.StringReceived THEN
		(* We have received a reply. Reset timers and triggers. *)
		fbTimer (IN := FALSE); 	(* reset timer *)

		statRef.sReply := CONCAT(statRef.sReply, DeviceReply);	(* CONCAT the reply *)
		nNumReplies	:= nNumReplies + 1;	(* Increment the number of replies *)

		IF nNumReplies = ctrlRef.nNumReplies THEN
			(* Clear the receive buffer ONLY when all replies have been received! *)
			ClearComBufferRx (Buffer := RxBuffer);
			State 			:= E_RS_COMM_STATE.IDLE;
			statRef.nStatus	:= E_RS_COMM_STATUS.IDLE;
			statRef.sStatus	:= 'IDLE';
		ELSE
			(* Stay in the same state and receive further replies *)
			;
		END_IF

		RETURN;

	END_IF



E_RS_COMM_STATE.CLEAR_BUFFER:
	(* Read any character present in the receive buffer *)
	(* 1 sec timeout for reply *)
	fbTimer (IN := TRUE, PT := T#1S);
	IF fbTimer.Q THEN
		(* reset timer *)
		fbTimer (IN := FALSE);
		statRef.bInitialised	:= TRUE;
		statRef.nStatus			:= E_RS_COMM_STATUS.IDLE;
		statRef.sStatus			:= 'INITIALISED';
		State 					:= E_RS_COMM_STATE.IDLE;
		RETURN;
	END_IF

	Receive(
		Prefix			:= '',
		Suffix			:= '',
		Timeout			:= T#500MS,
		ReceivedString	:= DeviceReply,
		RXbuffer		:= RxBuffer,
		Reset			:= FALSE);


ELSE
(* Unsuported state *)
	State 			:= E_RS_COMM_STATE.ERROR;
	statRef.nErrorCode	:= E_RS_COMM_ERROR.WRONG_STATE;
	statRef.sErrorText	:= 'Unknown State';
END_CASE

METHOD M_ActionInitExecute
VAR_INPUT
END_VAR
// TODO: Implement in extended FB
END_METHOD

METHOD M_ActivityConnect
VAR_INPUT
END_VAR
// TODO: Implement in extended FB
END_METHOD

METHOD M_ComPortControl
VAR_INPUT
END_VAR
// TODO: Implement in extended FB
END_METHOD

METHOD M_GetInitialised : BOOL
VAR_INPUT
END_VAR
M_GetInitialised	:= statRef.bInitialised;
END_METHOD

METHOD M_GetStatus : E_RS_COMM_STATUS
VAR_INPUT
END_VAR
M_GetStatus	:= statRef.nStatus;
END_METHOD

METHOD M_Reset
VAR_INPUT
END_VAR
// TODO: Implement in extended FB
END_METHOD

END_FUNCTION_BLOCK

// POUs/Comm/FB_RS_COMM_LAKESHORE
FUNCTION_BLOCK FB_RS_COMM_LAKESHORE EXTENDS FB_RS_COMM_BASE
VAR_INPUT
END_VAR
VAR_OUTPUT
END_VAR
VAR CONSTANT
END_VAR
VAR
	{attribute 'OPC.UA.DA' := '1'}
	cfg:		T_RS_COMM_CFG;				// Config parameters
	{attribute 'OPC.UA.DA' := '1'}
	ctrl:		T_RS_COMM_CTRL;				// Control parameters
	{attribute 'OPC.UA.DA' := '1'}
	{attribute 'OPC.UA.DA.Access' := '1'}
	info:		T_RS_COMM_INFO; 			// Info parameters - ReadOnly
	{attribute 'OPC.UA.DA' := '1'}
	{attribute 'OPC.UA.DA.Access' := '1'}
	stat:		T_RS_COMM_STAT;				// Status parameters - ReadOnly

	sim:		FB_SIM_RS_COMM_LAKESHORE;		// COMM simulator

	// Physical signals - to be mapped to EL60xx serial port controller !!!
	COMin_EL60xx	AT %I* 	: KL6inData22B;	(* linked to the EL60xx *)
	COMout_EL60xx	AT %Q*	: KL6outData22B;(* linked to the EL60xx *)

	(* Serial line control *)
	COMportControl: 		SerialLineControl;

END_VAR

// Set references
cfgRef	REF=cfg;
ctrlRef	REF=ctrl;
infoRef	REF=info;
statRef	REF=stat;
simRef	REF=sim;

SUPER^();

METHOD M_ActionInitExecute
VAR_INPUT
END_VAR
//
// Copy input parameters to cfg
//
cfg.sCmdSuffix		:= in_sCmdSuffix;
cfg.sReplySuffix	:= in_sReplySuffix;
cfg.nTimeout		:= in_nTimeout;

//
// If in simulation, there is no need to reset anything.
// Just set it to initialised and go to IDLE state.
//
IF in_bSimulation THEN
	fbTimer (IN := FALSE);
	statRef.bInitialised	:= TRUE;
	statRef.nStatus			:= E_RS_COMM_STATUS.IDLE;
	statRef.sStatus			:= 'INITIALISED';
	State 					:= E_RS_COMM_STATE.IDLE;
ELSE
	stat.bInitialised	:= FALSE;
	stat.sStatus		:= 'INITIALISING';
	stat.nStatus		:= E_RS_COMM_STATUS.BUSY;
	stat.sReply 		:= ''; (* No reply yet *)
	stat.nErrorCode		:= E_RS_COMM_ERROR.OK;
	stat.sErrorText		:= 'OK';
	
	// Reset the connected serial hardware 
	ComReset (
		Execute 	:= FALSE,
		pComIn		:= ADR(COMin_EL60xx),
		pComOut		:= ADR(COMout_EL60xx),
		SizeComIn	:= SIZEOF(COMin_EL60xx),
		);
	
	// Set next state
	State 	:= E_RS_COMM_STATE.RESET;
END_IF
END_METHOD

METHOD M_ComPortControl
VAR_INPUT
END_VAR
// RS specific call of the background communication process
COMportControl(
	Mode		:= ComSerialLineMode_t.SERIALLINEMODE_KL6_22B_STANDARD,
	pComIn		:= ADR(COMin_EL60xx),					(* I/O data; see global variables *)
	pComOut		:= ADR(COMout_EL60xx),					(* I/O data; see global variables *)
	SizeComIn	:= UINT_TO_INT(SIZEOF(COMin_EL60xx)),	(* I/O data; see global variables *)
	TxBuffer	:= TxBuffer,							(* transmit buffer; see global variables *)
	RxBuffer	:= RxBuffer);							(* receive buffer; see global variables *)
END_METHOD

METHOD M_Reset
VAR_INPUT
END_VAR
// RS specific call of communication reset
//
// Reset the connected serial hardware.
ComReset (
	Execute 	:= TRUE,
	pComIn		:= ADR(COMin_EL60xx),
	pComOut		:= ADR(COMout_EL60xx),
	SizeComIn	:= SIZEOF(COMin_EL60xx),
	);

(* Next step is to clear the buffers *)
IF ComReset.Done THEN
	fbTimer (IN := FALSE);	// Reset the timer
	State 		:= E_RS_COMM_STATE.CLEAR_BUFFER;
END_IF
END_METHOD

END_FUNCTION_BLOCK

// POUs/Comm/FB_RS_COMM_NO_SIM
FUNCTION_BLOCK FB_RS_COMM_NO_SIM EXTENDS FB_RS_COMM_BASE
VAR_INPUT
END_VAR
VAR_OUTPUT
END_VAR
VAR CONSTANT
END_VAR
VAR
	{attribute 'OPC.UA.DA' := '1'}
	cfg:		T_RS_COMM_CFG;				// Config parameters
	{attribute 'OPC.UA.DA' := '1'}
	ctrl:		T_RS_COMM_CTRL;				// Control parameters
	{attribute 'OPC.UA.DA' := '1'}
	{attribute 'OPC.UA.DA.Access' := '1'}
	info:		T_RS_COMM_INFO; 			// Info parameters - ReadOnly
	{attribute 'OPC.UA.DA' := '1'}
	{attribute 'OPC.UA.DA.Access' := '1'}
	stat:		T_RS_COMM_STAT;				// Status parameters - ReadOnly

	sim:		FB_SIM_RS_COMM_BASE;		// COMM simulator

	// Physical signals - to be mapped to EL60xx serial port controller !!!
	COMin_EL60xx	AT %I* 	: KL6inData22B;	(* linked to the EL60xx *)
	COMout_EL60xx	AT %Q*	: KL6outData22B;(* linked to the EL60xx *)

	(* Serial line control *)
	COMportControl: 		SerialLineControl;

END_VAR

// Set references
cfgRef	REF=cfg;
ctrlRef	REF=ctrl;
infoRef	REF=info;
statRef	REF=stat;
simRef	REF=sim;

SUPER^();

METHOD M_ActionInitExecute
VAR_INPUT
END_VAR
//
// Copy input parameters to cfg
//
cfg.sCmdSuffix		:= in_sCmdSuffix;
cfg.sReplySuffix	:= in_sReplySuffix;
cfg.nTimeout		:= in_nTimeout;

//
// If in simulation, there is no need to reset anything.
// Just set it to initialised and go to IDLE state.
//
IF in_bSimulation THEN
	fbTimer (IN := FALSE);
	statRef.bInitialised	:= TRUE;
	statRef.nStatus			:= E_RS_COMM_STATUS.IDLE;
	statRef.sStatus			:= 'INITIALISED';
	State 					:= E_RS_COMM_STATE.IDLE;
ELSE
	stat.bInitialised	:= FALSE;
	stat.sStatus		:= 'INITIALISING';
	stat.nStatus		:= E_RS_COMM_STATUS.BUSY;
	stat.sReply 		:= ''; (* No reply yet *)
	stat.nErrorCode		:= E_RS_COMM_ERROR.OK;
	stat.sErrorText		:= 'OK';
	
	// Reset the connected serial hardware 
	ComReset (
		Execute 	:= FALSE,
		pComIn		:= ADR(COMin_EL60xx),
		pComOut		:= ADR(COMout_EL60xx),
		SizeComIn	:= SIZEOF(COMin_EL60xx),
		);
	
	// Set next state
	State 	:= E_RS_COMM_STATE.RESET;
END_IF
END_METHOD

METHOD M_ComPortControl
VAR_INPUT
END_VAR
// RS specific call of the background communication process
COMportControl(
	Mode		:= ComSerialLineMode_t.SERIALLINEMODE_KL6_22B_STANDARD,
	pComIn		:= ADR(COMin_EL60xx),					(* I/O data; see global variables *)
	pComOut		:= ADR(COMout_EL60xx),					(* I/O data; see global variables *)
	SizeComIn	:= UINT_TO_INT(SIZEOF(COMin_EL60xx)),	(* I/O data; see global variables *)
	TxBuffer	:= TxBuffer,							(* transmit buffer; see global variables *)
	RxBuffer	:= RxBuffer);							(* receive buffer; see global variables *)
END_METHOD

METHOD M_Reset
VAR_INPUT
END_VAR
// RS specific call of communication reset
//
// Reset the connected serial hardware.
ComReset (
	Execute 	:= TRUE,
	pComIn		:= ADR(COMin_EL60xx),
	pComOut		:= ADR(COMout_EL60xx),
	SizeComIn	:= SIZEOF(COMin_EL60xx),
	);

(* Next step is to clear the buffers *)
IF ComReset.Done THEN
	fbTimer (IN := FALSE);	// Reset the timer
	State 		:= E_RS_COMM_STATE.CLEAR_BUFFER;
END_IF
END_METHOD

END_FUNCTION_BLOCK

// POUs/Comm/FB_USB_COMM_NO_SIM
FUNCTION_BLOCK FB_USB_COMM_NO_SIM EXTENDS FB_RS_COMM_BASE
VAR_INPUT
END_VAR
VAR_OUTPUT
END_VAR
VAR CONSTANT
END_VAR
VAR
	{attribute 'OPC.UA.DA' := '1'}
	cfg:		T_USB_COMM_CFG;				// Config parameters
	{attribute 'OPC.UA.DA' := '1'}
	ctrl:		T_RS_COMM_CTRL;				// Control parameters
	{attribute 'OPC.UA.DA' := '1'}
	{attribute 'OPC.UA.DA.Access' := '1'}
	info:		T_RS_COMM_INFO; 			// Info parameters - ReadOnly
	{attribute 'OPC.UA.DA' := '1'}
	{attribute 'OPC.UA.DA.Access' := '1'}
	stat:		T_RS_COMM_STAT;				// Status parameters - ReadOnly

	sim:		FB_SIM_RS_COMM_BASE;		// COMM simulator
	
	(* Serial line control *)
	SerialCfg: 				ComSerialConfig;
	COMportControl: 		SerialLineControlADS;

END_VAR

// Set references
cfgRef	REF=cfg;
ctrlRef	REF=ctrl;
infoRef	REF=info;
statRef	REF=stat;
simRef	REF=sim;

SUPER^();

METHOD M_ActionInitExecute
VAR_INPUT
END_VAR
stat.bInitialised	:= FALSE;
stat.sStatus		:= 'INITIALISING';
stat.nStatus		:= E_RS_COMM_STATUS.BUSY;
stat.sReply 		:= ''; (* No reply yet *)
stat.nErrorCode		:= E_RS_COMM_ERROR.OK;
stat.sErrorText		:= 'OK';

// Copy input parameters to cfg
cfg.sCmdSuffix		:= in_sCmdSuffix;
cfg.sReplySuffix	:= in_sReplySuffix;
cfg.nTimeout		:= in_nTimeout;

// Copy communication configuration
SerialCfg.ComPort	:= cfg.ComPort;
SerialCfg.Baudrate	:= cfg.Baudrate;
SerialCfg.DataBits	:= cfg.DataBits;
SerialCfg.Parity	:= cfg.Parity;
SerialCfg.StopBits	:= cfg.StopBits;

// Set next state
// Set 10 sec timeout for CONNECT, i.e. start the timer.
fbTimer(IN:=FALSE);
fbTimer(IN:=TRUE, PT:=T#10S);
State	:= E_RS_COMM_STATE.CONNECT;
END_METHOD

METHOD M_ActivityConnect
VAR_INPUT
END_VAR
// USB specific implementation of CONNECT
fbTimer();
IF fbTimer.Q THEN
	fbTimer(IN:=FALSE);
	State 			:= E_RS_COMM_STATE.ERROR;
	stat.nErrorCode	:= E_RS_COMM_ERROR.TIMEOUT;
	stat.sErrorText	:= 'Timeout on Port Open';
	RETURN;
END_IF

// Check if the port is open
IF COMportControl.PortOpened THEN
	State := E_RS_COMM_STATE.CLEAR_BUFFER;
END_IF
END_METHOD

METHOD M_ComPortControl
VAR_INPUT
END_VAR
// USB specific call of the background communication process
COMportControl(
	Connect		:= TRUE,		// Connect to serial port [TRUE=connect, FALSE=disconnect]
	SerialCfg	:= SerialCfg,	// Serial port configuration
	TxBuffer	:= TxBuffer,	// Serial Tx ComBuffer
	RxBuffer	:= RxBuffer);	// Serial Rx ComBuffer
END_METHOD

END_FUNCTION_BLOCK

// POUs/Devices/FB_CCC
FUNCTION_BLOCK FB_CCC EXTENDS FB_RS_BASE
VAR_INPUT
	{attribute 'OPC.UA.DA' := '0'}
	in_nPeriod:	DINT := 10000;	// Interval for periodic reading [ms], default 10000 ms = 10 sec 
END_VAR
VAR_OUTPUT
END_VAR
VAR CONSTANT
	{attribute 'OPC.UA.DA' := '0'}
	sCmdSuffix:		STRING(16) := '$0D';
	{attribute 'OPC.UA.DA' := '0'}
	sReplySuffix:	STRING(16) := '$0D';
END_VAR
VAR
	{attribute 'OPC.UA.DA' := '1'}
	cfg:		T_CCC_CFG;					//  Config parameters
	{attribute 'OPC.UA.DA' := '1'}
	ctrl:		T_CCC_CTRL;					//  Control parameters
	{attribute 'OPC.UA.DA' := '1'}
	{attribute 'OPC.UA.DA.Access' := '1'}
	info:		T_CCC_INFO; 				//  Info parameters - ReadOnly
	{attribute 'OPC.UA.DA' := '1'}
	{attribute 'OPC.UA.DA.Access' := '1'}
	stat:		T_CCC_STAT;					//  Status parameters - ReadOnly

	{attribute 'OPC.UA.DA' := '0'}
	comm:		FB_RS_COMM_NO_SIM;					// Instance of generic comm object. OPC UA Disabled!!!
	
	(* Pointers *)
	{attribute 'OPC.UA.DA' := '0'}
	ptrCommCfg:		POINTER TO T_RS_COMM_CFG 	:= ADR(comm.cfg);	(* Pointer to comm.cfg instance *)
	{attribute 'OPC.UA.DA' := '0'}
	ptrCommCtrl:	POINTER TO T_RS_COMM_CTRL 	:= ADR(comm.ctrl);	(* Pointer to comm.ctrl instance *)
	{attribute 'OPC.UA.DA' := '0'}
	ptrCommStat:	POINTER TO T_RS_COMM_STAT 	:= ADR(comm.stat);	(* Pointer to comm.stat instance *)
	{attribute 'OPC.UA.DA' := '0'}
	ptrInitCmds:	POINTER TO ARRAY [1..4] OF T_CCC_COMMAND;		(* Pointer to INIT commands *)
	{attribute 'OPC.UA.DA' := '0'}
	ptrReadCmds:	POINTER TO ARRAY [1..4] OF T_CCC_COMMAND;		(* Pointer to READ commands *)


	(* Timers *)
	{attribute 'OPC.UA.DA' := '0'}
	fbTimer:			TON; (* General Timeout *)
	
	(* Misc internal vars *)
	{attribute 'OPC.UA.DA' := '0'}
	cmdCounter:			INT := 1;

END_VAR

// Set references
cfgRef	REF=cfg;
ctrlRef	REF=ctrl;
statRef	REF=stat;


(* Execute comm instance *)
comm(in_sCmdSuffix:=sCmdSuffix, in_sReplySuffix:=sReplySuffix, in_nTimeout:=3000);


// Execute the base class object FB_RS_BASE
SUPER^();

METHOD ActivityInitializing
VAR_INPUT
	bExecute:	BOOL;
END_VAR
VAR_INST
	{attribute 'OPC.UA.DA' := '0'}
    nMethodState:	INT := 0;	// State Machine current state
END_VAR
SetAction('ActivityInitializing');


IF NOT bExecute THEN
	nMethodState	:= 0;	// Reset the state machine
	cmdCounter		:= 1;	// Init will start from the first init command
	RETURN;
END_IF

// Handle State Machine
CASE nMethodState OF
	0:	// Set communication parameters and Model configuration

		(* Set comm suffixes for commands and replies *)
		ptrCommCfg^.sCmdSuffix		:= sCmdSuffix;
		ptrCommCfg^.sReplySuffix	:= sReplySuffix;

		// Set monitoring period (input parameter)
		cfg.tDelay_Periodic	:= DINT_TO_TIME(in_nPeriod);
		// Auto monitor, i.e. monitor in Standby_Ready as well
		cfg.bAutoMonitor	:= TRUE;

		(* Set pointer to INIT and READ commands *)
		ptrInitCmds := ADR(cfg.cmdList_Init);
		ptrReadCmds := ADR(cfg.cmdList_Read);
		(* Set initial state and status *)
		stat.bInitialised	:= FALSE;
		stat.sReply			:= '';
		stat.sDeviceID		:= '';

		SetStatus(E_SM_ERROR.OK, 'BUSY');

		nMethodState := 10;				// Go to next state, i.e. INIT_COMM

	10:	// Initialize COMM port
		(* Reset the serial port *)
		ptrCommCtrl^.nCommand	:= E_RS_COMM_CMD.INIT;
		ptrCommCtrl^.bExecute	:= TRUE;

		// Init dev will start from the first init command.
		// We set counter to 0. It will be incremented in Wait IDLE.
		cmdCounter	:= 0;

		(* Start the timer by going false/true *)
		fbTimer (IN := FALSE); (* Reset timer *)
		fbTimer (IN := TRUE, PT := T#5S); (* 5 sec timeout for reply *)

		nMethodState 	:= 15;	// On next cycle wait until the comm port is reset, i.e. idle
		
	15:	// Wait IDLE
		fbTimer (IN := TRUE);
		IF comm.stat.nStatus = E_RS_COMM_STATUS.IDLE THEN
			// Communication is IDLE 
			fbTimer (IN := FALSE);	// disable timer 
			stat.sReply		:= ptrCommStat^.sReply;	// Save the reply

			IF cmdCounter >= 1 THEN
				// We are IDLE after an INIT command, i.e. CCC_CMD_RESET or CCC_CMD_GET_VERS
				IF ptrInitCmds^ [cmdCounter].cmd = cfg.CCC_CMD_RESET  THEN
					(* No action. Just check proper reply. *)
					IF FIND (stat.sReply, 'N')= 1 THEN
						SetStatus(E_CCC_ERROR.COMM, 'ERROR: Failed to RESET device');
						bCommProblem	:= TRUE;
						nEvent := E_SM_EVENT.ERRINIT;
						RETURN;
					END_IF
				ELSIF ptrInitCmds^ [cmdCounter].cmd = cfg.CCC_CMD_GET_VERS  THEN
					(* Save the reply into stat.sDeviceID. *)
					IF FIND (stat.sReply, 'N')= 1 THEN
						SetStatus(E_CCC_ERROR.COMM, 'ERROR: Command GET_VERS failed');
						bCommProblem	:= TRUE;
						nEvent := E_SM_EVENT.ERRINIT;
						RETURN;
					ELSIF FIND (stat.sReply, 'ESO')<> 2 THEN
						SetStatus(E_CCC_ERROR.COMM, 'ERROR: Failed to get device ID');
						bCommProblem	:= TRUE;
						nEvent := E_SM_EVENT.ERRINIT;
						RETURN;
					ELSE
						stat.sDeviceID	:= MID (stat.sReply, LEN(stat.sReply)-5, 2);
					END_IF
				END_IF
			END_IF

			// Restart the timer for delay between INIT commands
			fbTimer (IN := FALSE);	// disable timer 
			fbTimer (IN := TRUE, PT := cfg.tDelay_Init); // Wait INIT delay
			
			cmdCounter		:= cmdCounter + 1;	// Increment init command index
			bCommProblem	:= FALSE;
			nMethodState 	:= 18;	// Execute next device INIT command
		ELSIF comm.stat.nStatus = E_RS_COMM_STATUS.ERROR THEN
			fbTimer (IN := FALSE);
			SetStatus(E_CCC_ERROR.COMM, 'ERROR: Communication error');	
			bCommProblem	:= TRUE;
			nEvent := E_SM_EVENT.ERRINIT;
			RETURN;
		ELSIF fbTimer.Q THEN
			// Timer expired after 5 sec. This is an error.
			fbTimer (IN := FALSE);
			SetStatus(E_CCC_ERROR.TIMEOUT, 'ERROR: Communication timeout');	
			bCommProblem	:= TRUE;
			nEvent := E_SM_EVENT.ERRINIT;
			RETURN;
		END_IF

	
	
	18:	// Wait INIT Delay
		fbTimer (IN := TRUE);
		IF fbTimer.Q THEN
			// Timer expired after 5 sec. This is an error.
			fbTimer (IN := FALSE);
			nMethodState 	:= 20;	// Execute next device INIT command
			RETURN;
		END_IF

	
	
	20:	// INIT DEV
		IF ptrInitCmds^ [cmdCounter].cmd = '' THEN
			// Device INIT is done. Go to IDLE 
			stat.bInitialised 	:= TRUE;
			cmdCounter			:= 1;
			SetStatus(E_CCC_STATUS.IDLE, 'IDLE');
			nEvent 		:= E_SM_EVENT.INITDONE;
			RETURN;
		END_IF
		
		(* Send INIT command with index cmdCounter *)
		ptrCommCtrl^.nCommand		:= E_RS_COMM_CMD.SEND;
		ptrCommCtrl^.sCmd			:= ptrInitCmds^ [cmdCounter].cmd;
		ptrCommCtrl^.nNumReplies	:= 1;
		ptrCommCtrl^.bHasReply		:= TRUE;
		ptrCommCtrl^.bExecute		:= TRUE;
	
		(* Start the timer by going false/true *)
		fbTimer (IN := FALSE); (* Reset timer *)
		fbTimer (IN := TRUE, PT := T#5S); (* 5 sec timeout for reply *)

		// On next cycle wait until the comm port is idle
		nMethodState 	:= 15;	// On next cycle wait until the comm port is idle
	
END_CASE
END_METHOD

METHOD ActivityMonitoring
VAR_INPUT
	bExecute:	BOOL;
END_VAR
VAR_INST
	{attribute 'OPC.UA.DA' := '0'}
    nMethodState:	INT := 0;	// State Machine current state
	{attribute 'OPC.UA.DA' := '0'}
	nRetries:		INT := 0;	// Number of retries in case of communication problems
END_VAR
VAR
	bError:			BOOL;
END_VAR
IF NOT bExecute THEN
	SetAction('ActivityMonitoring'); 
	SetStatus(E_SM_ERROR.OK, 'BUSY');
	nMethodState	:= 0;	// Reset the state machine
	cmdCounter		:= 1;	// Reading will start from the first command in the array
	nRetries		:= 0;					
	RETURN;
END_IF

// Handle State Machine
CASE nMethodState OF
	0:	// Execute a command from the command array
		IF ptrReadCmds^ [cmdCounter].cmd = '' OR cmdCounter > 4 THEN
			// We arrived to the end of the array of pre-defined commands
			// Check if we have to exit Monitoring
			IF nNextState <> E_RS_BASE_STATE.NONE	THEN
				SetStatus(E_SM_ERROR.OK, nNextDescription);
				SetState(nNextState, nNextSubstate);
				nNextState		:= E_RS_BASE_STATE.NONE;
				nNextSubstate	:= E_RS_BASE_SUBSTATE.NONE;
				nNextDescription:= 'IDLE';
				RETURN;
			END_IF

			// Periodic READ is done. Wait tDelay_Periodic before re-starting the READ.
			cmdCounter	:= 1;
			SetStatus(E_SM_ERROR.OK, 'IDLE');
			
			(* Start the timer by going false/true *)
			fbTimer (IN := FALSE); (* Reset timer *)
			fbTimer (IN := TRUE, PT := cfg.tDelay_Periodic);
			nMethodState := 10;				// Goto Wait for tDelay_Periodic
			RETURN;
		END_IF
		
		(* Send command with index cmdCounter *)
		ptrCommCtrl^.nCommand		:= E_RS_COMM_CMD.SEND;
		ptrCommCtrl^.sCmd			:= ptrReadCmds^ [cmdCounter].cmd;
		ptrCommCtrl^.nNumReplies	:= 1;
		ptrCommCtrl^.bHasReply		:= TRUE;
		ptrCommCtrl^.bExecute		:= TRUE;
		
		stat.sErrorText := 'BUSY';
		(* Start the timer by going false/true *)
		fbTimer (IN := FALSE); (* Reset timer *)
		fbTimer (IN := TRUE, PT := T#5S); (* 5 sec timeout for reply *)

		nMethodState := 20;				// Goto WAIT for Reading to complete,

	10:	// Wait until the delay timeout expires
		fbTimer (IN := TRUE);

		// Check if we have to exit Monitoring
		IF nNextState <> E_RS_BASE_STATE.NONE THEN
			fbTimer (IN := FALSE); (* Stop the timer *)
			SetStatus(E_SM_ERROR.OK, nNextDescription);
			SetState(nNextState, nNextSubstate);
			nNextState		:= E_RS_BASE_STATE.NONE;
			nNextSubstate	:= E_RS_BASE_SUBSTATE.NONE;
			nNextDescription:= 'IDLE';
			RETURN;
		END_IF
	
		(* If Timer has expired, go to the next state. *)
		IF fbTimer.Q THEN
			fbTimer (IN := FALSE);
			cmdCounter		:= 1;	// Reading will start from the first command in the array
			nMethodState 	:= 0;	// Goto Wait for tDelay_Periodic
			RETURN;
		END_IF
	


	20:	// Wait for the reading to complete, i.e. IDLE
		fbTimer (IN := TRUE);
		IF comm.stat.nStatus = E_RS_COMM_STATUS.IDLE THEN
			bError	:= FALSE;
			// Communication is IDLE 
			fbTimer (IN := FALSE);	// disable timer 
			stat.sReply		:= ptrCommStat^.sReply;	// Save the reply
			
			(* Extract the readins from the reply. *)
			IF ptrReadCmds^ [cmdCounter].cmd = cfg.CCC_CMD_GET_STAT  THEN
				IF NOT M_UpdateDevStatus() THEN
					SetStatus(E_CCC_ERROR.COMM, 'ERROR: GET_STAT reply format not correct');
					bError	:= TRUE;
				END_IF
			ELSIF ptrReadCmds^ [cmdCounter].cmd = cfg.CCC_CMD_GET_TEMP  THEN
				IF NOT M_UpdateDevTemps() THEN
					SetStatus(E_CCC_ERROR.COMM, 'ERROR: GET_TEMP reply format not correct');
					bError	:= TRUE;
				END_IF
			ELSIF ptrReadCmds^ [cmdCounter].cmd = cfg.CCC_CMD_GET_FLOW  THEN
				IF NOT M_UpdateDevFlows() THEN
					SetStatus(E_CCC_ERROR.COMM, 'ERROR: GET_FLOW reply format not correct');
					bError	:= TRUE;
				END_IF
			END_IF

			bCommProblem	:= FALSE;
			nRetries		:= 0;	// Reset number of retries
			
			// Check if we have to exit Monitoring
			IF nNextState <> E_RS_BASE_STATE.NONE THEN
				fbTimer (IN := FALSE); (* Stop the timer *)
				SetStatus(E_SM_ERROR.OK, nNextDescription);
				SetState(nNextState, nNextSubstate);
				nNextState		:= E_RS_BASE_STATE.NONE;
				nNextSubstate	:= E_RS_BASE_SUBSTATE.NONE;
				nNextDescription:= 'IDLE';
				RETURN;
			END_IF
	
			cmdCounter		:= cmdCounter + 1;	// Reading will start from the first command in the array
			
			nMethodState 	:= 0;				// Goto Send command
			nEvent := E_SM_EVENT.COMMOK;
			RETURN;
		ELSIF comm.stat.nStatus = E_RS_COMM_STATUS.ERROR OR fbTimer.Q THEN
			fbTimer (IN := FALSE);
			SetStatus(E_CCC_ERROR.COMM, 'ERROR: Communication error');	
			bCommProblem	:= TRUE;
			// Retry up to 2 times
			nRetries		:= nRetries + 1;		// Increment number of retries
			stat.nRetries	:= stat.nRetries + 1;	// Increment total number of retries
			IF nRetries > 1 THEN
				nEvent := E_SM_EVENT.ERRCOMM;
			END_IF
			// Apply a short delay of 1 sec and retry
			fbTimer (IN := FALSE); (* Reset timer *)
			fbTimer (IN := TRUE, PT := T#1000MS);
			nMethodState := 10;				// Goto Wait 
			RETURN;
		ELSIF bError THEN
			// Apply a short delay of 3 sec and retry
			fbTimer (IN := FALSE); (* Reset timer *)
			fbTimer (IN := TRUE, PT := T#3000MS);
			nMethodState := 10;				// Goto Wait 
			RETURN;
		END_IF

	
END_CASE
END_METHOD

METHOD M_ConvertTemp : LREAL
VAR_INPUT
	lrTempNorm:	WORD;	(* Normalised temperature *)
END_VAR
M_ConvertTemp	:= (WORD_TO_LREAL(lrTempNorm) - 5750) / 375.0;
END_METHOD

METHOD M_SetAllFaulty : BOOL
(* 
	Method to set all readings to faulty, i.e. 9999.
	Used when communication fails.
*)
VAR_INPUT
END_VAR
VAR_OUTPUT
END_VAR
VAR
END_VAR
stat.bWarn_relay2_alarm	:= TRUE;

stat.lrTemp_outlet	:= 9999;
stat.lrTemp_inlet	:= 9999;
stat.lrTemp_cabinet	:= 9999;
stat.lrTemp_ambient	:= 9999;

stat.lrFlow_1	:= 9999;
stat.lrFlow_2	:= 9999;
stat.lrFlow_3	:= 9999;

M_SetAllFaulty	:= TRUE;
END_METHOD

METHOD M_TrimDevReply : BOOL
(* 
	 *
	 * reply syntax is:
	 * <init char><parameters><checksum><end char>
	 * whereby
	 * init char = 'A' for OK or 'N' for ERROR.
	 * parameters = reply body for reply OK or <error code> for error
	 * checksum, 2 chars
	 * end char = <CR> (but there is also another undocumented char in the reply)
	 
	 We want to extract <parameters>. We start from the 2nd char and take LEN-5 chars.
*)

VAR_INPUT
	sReply:	STRING;		(* Device reply string *)
END_VAR
VAR_OUTPUT
	sTrimmedString:	STRING;
END_VAR

VAR
END_VAR
(* If the first char is 'N', this is an error reply. *)
IF FIND (sReply, 'N')= 1 THEN
	sTrimmedString	:= '';
	M_TrimDevReply	:= FALSE;
	RETURN;
END_IF

(* Remove the first char and the last 3 chars *)
sTrimmedString := MID (sReply, LEN(sReply)-5, 2);
M_TrimDevReply	:= TRUE;
RETURN;
END_METHOD

METHOD M_UpdateDevFlows : BOOL
(* 
	Method to extract CCC device flow rates
	from the reply to command cfg.CCC_CMD_GET_FLOW, i.e. '>00f'.
	
         Body of reply to GET_TEMP command is:
         * flow rate #1 (main flow)	- 4 chars
         * flow rate #2 (main flow)	- 4 chars
         * flow rate #3 (main flow)	- 4 chars
         
	Reply is in HEX format !!!
	
*)

VAR_INPUT
END_VAR
VAR
	bOK:	BOOL;		(* TRUE if the reading was correct, i.e. 'n' values successfully extracted from 'str'.  *)
	
	sTrimmedReply:	STRING;
    data: 	ARRAY[0..5] OF WORD;
    cbData: UDINT;
	nWord:	WORD;

END_VAR
(* Trim the reply *)
bOK := M_TrimDevReply(sReply := stat.sReply, sTrimmedString => sTrimmedReply);

(* We are expecting 3 4-char strings (hex words) in the reply (6 bytes) *)
cbData := HEXSTR_TO_DATA (sTrimmedReply, ADR( data ), SIZEOF( data ));

IF NOT bOK  OR  cbData <> 6 THEN
	sTrimmedReply	:= '';
	M_UpdateDevFlows	:= FALSE;
	RETURN;
END_IF

stat.lrFlow_1	:= WORD_TO_LREAL(HOST_TO_BE16 (data[0]));
stat.lrFlow_2	:= WORD_TO_LREAL(HOST_TO_BE16 (data[1]));
stat.lrFlow_3	:= WORD_TO_LREAL(HOST_TO_BE16 (data[2]));


M_UpdateDevFlows	:= TRUE;
END_METHOD

METHOD M_UpdateDevStatus : BOOL
(* 
	Method to extract CCC device status from the 
	reply to command cfg.CCC_CMD_GET_STAT, i.e. '>00o'.
	
         Body of reply to GET_STAT command is:
         * <CSTAT1> 				- 2 chars
         * <CSTAT2> 				- 2 chars
         * <feprom status> 			- 2 chars
         * <communication status> 	- 2 chars
         * <debugr> 				- 2 chars
         
	Reply is in HEX format !!!
	We use only <CSTAT1> and <CSTAT2>.
	
*)

VAR_INPUT
END_VAR
VAR
	bOK:		BOOL;		(* TRUE if the reading was correct, i.e. 'n' values successfully extracted from 'str'.  *)
	
	sTrimmedReply:	STRING;
    data    : ARRAY[0..5] OF BYTE;
    cbData  : UDINT;
	bByte:	BYTE;

END_VAR
(* Trim the reply *)
bOK := M_TrimDevReply(sReply := stat.sReply, sTrimmedString => sTrimmedReply);

(* We are expecting 5 2-char strings in the reply *)
cbData := HEXSTR_TO_DATA (sTrimmedReply, ADR( data ), SIZEOF( data ));

IF NOT bOK  OR  cbData <> 5 THEN
	sTrimmedReply	:= '';
	M_UpdateDevStatus	:= FALSE;
	RETURN;
END_IF

(*
	<CSTAT1> = data [0]
	<CSTAT2> = data [1]
*)

(* Handling of <CSTAT1>, i.e. data[0] *)
stat.bWarn_cabinet_high			:= (data[0] AND 16#0001) <> 0;
stat.bWarn_cabinet_no_control	:= (data[0] AND 16#0002) <> 0;

IF (data[0] AND 16#0010) <> 0  THEN
	(* Warning code bit4 is active. Check bit2-3 for meaning. *) 
	bByte	:= (SHL(data[0],2) AND 16#0003);
	CASE bByte OF
	0:	stat.bWarn_outlet_high			:= TRUE;
	1:	stat.bWarn_inlet_high			:= TRUE;
	2:	stat.bWarn_airflow_insufficient	:= TRUE;
	3:	stat.bWarn_coolant_insufficient	:= TRUE;
	END_CASE
ELSE
	stat.bWarn_outlet_high			:= FALSE;
	stat.bWarn_inlet_high			:= FALSE;
	stat.bWarn_airflow_insufficient	:= FALSE;
	stat.bWarn_coolant_insufficient	:= FALSE;
END_IF

stat.bWarn_door_open			:= (data[0] AND 16#0020) = 0;
stat.bWarn_relay1_warning		:= (data[0] AND 16#0040) <> 0;
stat.bWarn_relay2_alarm			:= (data[0] AND 16#0080) <> 0;


(* Handling of <CSTAT2>, i.e. data[1] *)
stat.bFault_temp_sensor_ambient	:= (data[1] AND 16#0001) <> 0;
stat.bFault_temp_sensor_cabinet	:= (data[1] AND 16#0002) <> 0;
stat.bFault_temp_sensor_inlet	:= (data[1] AND 16#0004) <> 0;
stat.bFault_temp_sensor_outlet	:= (data[1] AND 16#0008) <> 0;
stat.bFault_analog_supply		:= (data[1] AND 16#0040) <> 0;
stat.bFault_digital_supply		:= (data[1] AND 16#0080) <> 0;

M_UpdateDevStatus	:= TRUE;
END_METHOD

METHOD M_UpdateDevTemps : BOOL
(* 
	Method to extract CCC device temperatures and the main flow rate
	from the reply to command cfg.CCC_CMD_GET_TEMP, i.e. '>00H'.
	
         Body of reply to GET_TEMP command is:
         * flow rate #2 (main flow)	- 4 chars (ignored !!! Will be read with GET_FLOW)
         * <outlet temperature> 	- 4 chars
         * <inlet temperature> 		- 4 chars
         * <cabinet temperature> 	- 4 chars
         * <ambient temperature> 	- 4 chars
         
		 Temperatures are normalised. Real temperature is calculated as:
		 	Celsius = (TN - 5750)/375 
		 
	Reply is in HEX format !!!
	
*)

VAR_INPUT
END_VAR
VAR
	bOK:	BOOL;		(* TRUE if the reading was correct, i.e. 'n' values successfully extracted from 'str'.  *)
	
	sTrimmedReply:	STRING;
    data: 	ARRAY[0..5] OF WORD;
    cbData: UDINT;
	nWord:	WORD;

END_VAR
(* Trim the reply *)
bOK := M_TrimDevReply(sReply := stat.sReply, sTrimmedString => sTrimmedReply);

(* We are expecting 5 4-char strings (hex words) in the reply (10 bytes) *)
cbData := HEXSTR_TO_DATA (sTrimmedReply, ADR( data ), SIZEOF( data ));

IF NOT bOK  OR  cbData <> 10 THEN
	sTrimmedReply	:= '';
	M_UpdateDevTemps	:= FALSE;
	RETURN;
END_IF

(*	Before calculating the temperature, check for sensor failure.
	In case of sensor failure, set the value to the magic number 9999.
	Generic GUI's understand this as N/A, i.e. error or simulation. *)
IF stat.bFault_temp_sensor_outlet THEN
	stat.lrTemp_outlet	:= 9999;
ELSE
	stat.lrTemp_outlet	:= M_ConvertTemp(HOST_TO_BE16 (data[1]));
END_IF

IF stat.bFault_temp_sensor_inlet THEN
	stat.lrTemp_inlet	:= 9999;
ELSE
	stat.lrTemp_inlet	:= M_ConvertTemp(HOST_TO_BE16 (data[2]));
END_IF

IF stat.bFault_temp_sensor_cabinet THEN
	stat.lrTemp_cabinet	:= 9999;
ELSE
	stat.lrTemp_cabinet	:= M_ConvertTemp(HOST_TO_BE16 (data[3]));
END_IF

IF stat.bFault_temp_sensor_ambient THEN
	stat.lrTemp_ambient	:= 9999;
ELSE
	stat.lrTemp_ambient	:= M_ConvertTemp(HOST_TO_BE16 (data[4]));
END_IF


M_UpdateDevTemps	:= TRUE;
END_METHOD

END_FUNCTION_BLOCK

// POUs/MAIN
PROGRAM MAIN
VAR
	MCHR:	FB_RS_COMM_NO_SIM;
	PICO:	FB_RS_COMM_NO_SIM;

	{attribute 'OPC.UA.DA' := '1'}
	CCC:	FB_CCC;


	BBDY1:	FB_MODBUS_COMM_NO_SIM;
	
	{attribute 'OPC.UA.DA' := '1'}
	JUMO:	FB_JUMO;
	
	// Lakeshore 340 (RS-232 interface)
	{attribute 'OPC.UA.DA' := '1'}
	LS340:			FB_LAKESHORE_RS;


END_VAR

MCHR(in_sCmdSuffix:='$0D$0A',in_sReplySuffix:='>', in_nTimeout:=30000);
PICO(in_sCmdSuffix:='$0D',in_sReplySuffix:='$0D', in_nTimeout:=5000);

CCC(in_sName:='CCC', in_nPeriod := 1200);

BBDY1();

JUMO(in_sName:='JUMO',in_nPeriod:=1000);	// Read all JUMOs every second


LS340(	in_bSimulation		:= TRUE,		
		in_sName			:= 'Lake 340', 
		in_nModel			:= 340, 
		in_bAutoMonitor		:= TRUE,
		in_sCmdSuffix		:= '$0D$0A',
		in_sReplySuffix		:= '$0D$0A',
		in_nPeriod			:= 1700);

END_PROGRAM

// POUs/Devices/FB_JUMO
FUNCTION_BLOCK FB_JUMO EXTENDS FB_RS_BASE
VAR_INPUT
	{attribute 'OPC.UA.DA' := '0'}
	in_nPeriod:	DINT := 10000;	//Interval for periodic reading [ms], default 10000 ms = 10 sec
END_VAR
VAR_OUTPUT
END_VAR
VAR CONSTANT
END_VAR
VAR
	{attribute 'OPC.UA.DA' := '1'}
	cfg:		T_JUMO_CFG;					//  Config parameters
	{attribute 'OPC.UA.DA' := '1'}
	ctrl:		T_JUMO_CTRL;				//  Control parameters
	{attribute 'OPC.UA.DA' := '1'}
	{attribute 'OPC.UA.DA.Access' := '1'}
	info:		T_JUMO_INFO; 				//  Info parameters - ReadOnly
	{attribute 'OPC.UA.DA' := '1'}
	{attribute 'OPC.UA.DA.Access' := '1'}
	stat:		T_JUMO_STAT;				//  Status parameters - ReadOnly

	{attribute 'OPC.UA.DA' := '0'}
	comm:		FB_MODBUS_COMM_JUMO;		// Instance of generic comm object. OPC UA Disabled!!!
	
	(* Pointers *)
	{attribute 'OPC.UA.DA' := '0'}
	ptrCommCfg:		POINTER TO T_MODBUS_CFG 	:= ADR(comm.cfg);	(* Pointer to comm.cfg instance *)
	{attribute 'OPC.UA.DA' := '0'}
	ptrCommCtrl:	POINTER TO T_MODBUS_CTRL 	:= ADR(comm.ctrl);	(* Pointer to comm.ctrl instance *)
	{attribute 'OPC.UA.DA' := '0'}
	ptrCommStat:	POINTER TO T_MODBUS_STAT 	:= ADR(comm.stat);	(* Pointer to comm.stat instance *)


	(* Timers *)
	{attribute 'OPC.UA.DA' := '0'}
	fbTimer:			TON; (* General Timeout *)

END_VAR

// Set references
cfgRef	REF=cfg;
ctrlRef	REF=ctrl;
statRef	REF=stat;


(* Execute comm instance *)
comm(	in_bSimulation	:= in_bSimulation,
		in_nModel		:= 0,
		in_cReadFunction:= 3);


// Execute the base class object FB_RS_BASE
SUPER^();

METHOD ActivityInitializing
VAR_INPUT
	bExecute:	BOOL;
END_VAR
VAR_INST
	{attribute 'OPC.UA.DA' := '0'}
    nMethodState:	INT := 0;	// State Machine current state
END_VAR
VAR
	nInt:	INT;	// Temporary INT for conversion of ENUM types
END_VAR
SetAction('ActivityInitializing');


IF NOT bExecute THEN
	nMethodState	:= 0;	// Reset the state machine
	RETURN;
END_IF

// Handle State Machine
CASE nMethodState OF
	0:	// Set communication parameters and Model configuration


		// Set monitoring period (input parameter)
		cfg.tDelay_Periodic	:= DINT_TO_TIME(in_nPeriod);
		// Auto monitor, i.e. monitor in Standby_Ready as well
		cfg.bAutoMonitor	:= TRUE;

		(* Set initial state and status *)
		stat.bInitialised	:= FALSE;
		stat.nRetries		:= 0;

		SetStatus(E_SM_ERROR.OK, 'BUSY');
		
		// User configuration of the system
		M_UserConfigure();

		nMethodState := 10;				// Go to next state, i.e. INIT_COMM

	10:	// Initialize COMM port
		(* Reset the serial port *)
		nInt	:= E_RS_COMM_CMD.INIT;
		ptrCommCtrl^.nCommand	:= nInt;
		ptrCommCtrl^.bExecute	:= TRUE;

		(* Start the timer by going false/true *)
		fbTimer (IN := FALSE); (* Reset timer *)
		fbTimer (IN := TRUE, PT := T#5S); (* 5 sec timeout for reply *)

		nMethodState 	:= 15;	// On next cycle wait until the comm port is reset, i.e. idle
		
	15:	// Wait IDLE
		fbTimer (IN := TRUE);
		IF comm.stat.nStatus = E_RS_COMM_STATUS.IDLE THEN
			// Communication is IDLE 
			fbTimer (IN := FALSE);	// disable timer 
			stat.nInputBuffer		:= ptrCommStat^.DeviceReply;	// Save the reply

			bCommProblem	:= FALSE;
			// Device INIT is done. Go to IDLE 
			stat.bInitialised 	:= TRUE;
			SetStatus(E_CCC_STATUS.IDLE, 'IDLE');
			nEvent 		:= E_SM_EVENT.INITDONE;
			RETURN;
		ELSIF comm.stat.nStatus = E_RS_COMM_STATUS.ERROR THEN
			fbTimer (IN := FALSE);
			SetStatus(E_CCC_ERROR.COMM, 'ERROR: Communication error');	
			bCommProblem	:= TRUE;
			nEvent := E_SM_EVENT.ERRINIT;
			RETURN;
		ELSIF fbTimer.Q THEN
			// Timer expired after 5 sec. This is an error.
			fbTimer (IN := FALSE);
			SetStatus(E_CCC_ERROR.TIMEOUT, 'ERROR: Communication timeout');	
			bCommProblem	:= TRUE;
			nEvent := E_SM_EVENT.ERRINIT;
			RETURN;
		END_IF

	
	
	
END_CASE
END_METHOD

METHOD ActivityMonitoring
VAR_INPUT
	bExecute:	BOOL;
END_VAR
VAR_INST
	{attribute 'OPC.UA.DA' := '0'}
    nMethodState:	INT := 0;					// State Machine current state
	{attribute 'OPC.UA.DA' := '0'}
	nAddressIndex:	INT := E_JUMO_ADDRESS.COMMON;	// Which address space to read
	{attribute 'OPC.UA.DA' := '0'}
	nSlaveIndex:	INT := 1;
	{attribute 'OPC.UA.DA' := '0'}
	nRetries:		INT := 0;					// Number of retries in case of communication problems
END_VAR
IF NOT bExecute THEN
	SetAction('ActivityMonitoring'); 
	SetStatus(E_SM_ERROR.OK, 'BUSY');
	nMethodState	:= 0;	// Reset the state machine
	nSlaveIndex		:= M_GetFirstSlaveIndex();
	nAddressIndex	:= E_JUMO_ADDRESS.COMMON;
	ctrl.nSlaveID	:= cfg.aSlaveID[nSlaveIndex];
	ctrl.nRegister	:= cfg.nAddrCommon;
	ctrl.nWords		:= cfg.nWordsCommon;
	nRetries		:= 0;					
	RETURN;
END_IF

// Handle State Machine
CASE nMethodState OF
	0:	// Execute a command from the command array
		// Check if we have to exit Monitoring
		IF nNextState <> E_RS_BASE_STATE.NONE	THEN
			SetStatus(E_SM_ERROR.OK, nNextDescription);
			SetState(nNextState, nNextSubstate);
			nNextState		:= E_RS_BASE_STATE.NONE;
			nNextSubstate	:= E_RS_BASE_SUBSTATE.NONE;
			nNextDescription:= 'IDLE';
			RETURN;
		END_IF
		
		
		// Send command
		ptrCommCtrl^.nCommand		:= E_MODBUS_CMD.SEND;
		ptrCommCtrl^.nSlaveID		:= ctrl.nSlaveID;
		ptrCommCtrl^.nRegister		:= ctrl.nRegister;
		ptrCommCtrl^.nWords			:= ctrl.nWords;
		ptrCommCtrl^.bExecute		:= TRUE;
		
		(* Start the timer by going false/true *)
		fbTimer (IN := FALSE); (* Reset timer *)
		fbTimer (IN := TRUE, PT := T#5S); (* 5 sec timeout for reply *)

		nMethodState := 20;				// Goto WAIT for Reading to complete,

	10:	// Wait until the delay timeout expires
		fbTimer (IN := TRUE);

		// Check if we have to exit Monitoring
		IF nNextState <> E_RS_BASE_STATE.NONE THEN
			fbTimer (IN := FALSE); (* Stop the timer *)
			SetStatus(E_SM_ERROR.OK, nNextDescription);
			SetState(nNextState, nNextSubstate);
			nNextState		:= E_RS_BASE_STATE.NONE;
			nNextSubstate	:= E_RS_BASE_SUBSTATE.NONE;
			nNextDescription:= 'IDLE';
			RETURN;
		END_IF
	
		(* If Timer has expired, go to the next state. *)
		IF fbTimer.Q THEN
			fbTimer (IN := FALSE);
			SetStatus(E_SM_ERROR.OK, 'BUSY');
			nMethodState 	:= 0;	// Goto next reading
			RETURN;
		END_IF
	


	20:	// Wait for the reading to complete, i.e. IDLE
		fbTimer (IN := TRUE);
		IF comm.stat.nStatus = E_RS_COMM_STATUS.IDLE THEN
			// Communication is IDLE  
			fbTimer (IN := FALSE);	// disable timer 
			stat.nInputBuffer		:= ptrCommStat^.DeviceReply;	// Save the reply
			
			// Extract the readings from the reply.
			M_ExtractReadings(nSlaveIndex,nAddressIndex);

			bCommProblem	:= FALSE;
			nRetries		:= 0;	// Reset number of retries
			
			// Check if we have to exit Monitoring
			IF nNextState <> E_RS_BASE_STATE.NONE THEN
				fbTimer (IN := FALSE); (* Stop the timer *)
				SetStatus(E_SM_ERROR.OK, nNextDescription);
				SetState(nNextState, nNextSubstate);
				nNextState		:= E_RS_BASE_STATE.NONE;
				nNextSubstate	:= E_RS_BASE_SUBSTATE.NONE;
				nNextDescription:= 'IDLE';
				RETURN;
			END_IF
	
			IF NOT M_SetCommand(nSlaveIndex,nAddressIndex) THEN
				// We completed a full read cycle.
				// Wait periodic delay.
				// Periodic READ is done. Wait tDelay_Periodic before re-starting the READ.
				SetStatus(E_SM_ERROR.OK, 'IDLE');
				(* Start the timer by going false/true *)
				fbTimer (IN := FALSE); (* Reset timer *)
				fbTimer (IN := TRUE, PT := cfg.tDelay_Periodic);
				nMethodState := 10;				// Goto Wait 
				RETURN;
			ELSE
				// Apply a short delay of 30 ms after each command
				fbTimer (IN := FALSE); (* Reset timer *)
				fbTimer (IN := TRUE, PT := T#30MS);
				nMethodState := 10;				// Goto Wait 
				RETURN;
			END_IF

		ELSIF INT_TO_DINT(comm.stat.nStatus) = INT_TO_DINT(E_MODBUS_STATUS.ERROR) OR fbTimer.Q THEN
			fbTimer (IN := FALSE);
			SetStatus(E_MODBUS_ERROR.RECEIVE, 'ERROR: Communication error');	
			bCommProblem	:= TRUE;
			// Retry up to 3 times
			nRetries		:= nRetries + 1;		// Increment number of retries
			stat.nRetries	:= stat.nRetries + 1;	// Increment total number of retries
			IF nRetries > 3 THEN
				nEvent := E_SM_EVENT.ERRCOMM;
			ELSE
				// Apply a short delay of 1 sec and retry
				fbTimer (IN := FALSE); (* Reset timer *)
				fbTimer (IN := TRUE, PT := T#1000MS);
				nMethodState := 10;				// Goto Wait 
			END_IF
			RETURN;
		END_IF

	
END_CASE
END_METHOD

METHOD M_ByteSwapFLOAT : REAL
VAR_INPUT
	pByte:		POINTER TO BYTE;	// Pointer to array of bytes read from JUMO
END_VAR
VAR
	rResult:	REAL;
	pResult:	POINTER TO BYTE	:= ADR(rResult);	// Pointer to the result
END_VAR
pResult[0]	:= pByte[1];
pResult[1]	:= pByte[0];
pResult[2]	:= pByte[3];
pResult[3]	:= pByte[2];

M_ByteSwapFLOAT	:= rResult;
END_METHOD

METHOD M_ByteSwapINT : INT
VAR_INPUT
	pByte:		POINTER TO BYTE;	// Pointer to array of bytes read from JUMO
END_VAR
VAR
	nResult:	INT;
	pResult:	POINTER TO BYTE	:= ADR(nResult);	// Pointer to the result
END_VAR
pResult[0]	:= pByte[1];
pResult[1]	:= pByte[0];

M_ByteSwapINT	:= nResult;
END_METHOD

METHOD M_ExtractReadings : BOOL
VAR_INPUT
	nSlaveIndex:	INT;
	nAddressIndex:	INT;	// Which address space to read
END_VAR
VAR
	pBuf:	POINTER TO BYTE	:= ADR(stat.nInputBuffer);
	loop:	INT;
	par:	INT;
END_VAR
// There are 3 bytes before data starts !!!
IF nAddressIndex = E_JUMO_ADDRESS.COMMON THEN
	////////////////////////////
	// Extract Common Parameters
	////////////////////////////

	// Sampling time
	// Offset 3 + 0 = 3
	stat.aSamplingTime[nSlaveIndex]	:= M_ByteSwapFLOAT(ADR(pBuf[3]));

	// Internal PT100 temperature [degC]
	// Offset 3 + 4 = 7
	stat.aInternalTemperature[nSlaveIndex]	:= M_ByteSwapFLOAT(ADR(pBuf[7]));

	// - Analog Inputs
	// Offset 3 + 8 = 11
	FOR par := 1 TO 8 DO
		stat.aAnalogInputs[nSlaveIndex,par] := M_ByteSwapFLOAT(ADR(pBuf[11 + 4*(par-1)]));
	END_FOR

	// - Math
	// Offset 3 + 8 + 8*4 = 43
	FOR par := 1 TO 8 DO
		stat.aMath[nSlaveIndex,par] := M_ByteSwapFLOAT(ADR(pBuf[43 + 4*(par-1)]));
	END_FOR

	// Control Parameters
	// Offset 3 + 8 + 8*4 + 8*4 = 75
	FOR loop := 1 TO 4 DO
		FOR par := 1 TO 9 DO
			stat.aCtrlParams[nSlaveIndex,loop,par] := M_ByteSwapFLOAT(ADR(pBuf[75 + 40*(loop-1) + 4*(par-1)]));
		END_FOR
	END_FOR

	// - Switch Stats
	// Offset 3 + 8 + 8*4 + 8*4 + 9*4 = 111
	FOR loop := 1 TO 4 DO
		FOR par := 1 TO 2 DO
			stat.aSwitchStats[nSlaveIndex,loop,par] := M_ByteSwapINT(ADR(pBuf[111 + 40*(loop-1) + 2*(par-1)]));
		END_FOR
	END_FOR
ELSIF nAddressIndex = E_JUMO_ADDRESS.SET_POINTS THEN
	// Extract Set Points
	// Offset 3 + 0 = 3
	FOR loop := 1 TO 4 DO
		FOR par := 1 TO 4 DO
			stat.aSetPoints[nSlaveIndex,loop,par] := M_ByteSwapFLOAT(ADR(pBuf[3 + 16*(loop-1) + 4*(par-1)]));
		END_FOR
	END_FOR
END_IF
END_METHOD

METHOD M_GetFirstSlaveIndex : INT
VAR_INPUT
END_VAR
VAR
	i:	INT;
END_VAR
M_GetFirstSlaveIndex	:= i;
FOR i := 1 TO 8 DO
	IF cfg.aDevUsed[i] THEN
		M_GetFirstSlaveIndex	:= i;
		RETURN;
	END_IF
END_FOR
END_METHOD

METHOD M_GetNextSlaveIndex : INT
VAR_INPUT
	nSlaveIndex:	INT;
END_VAR
VAR
	i:	INT;
END_VAR
// Find the index if the next Used Slave.
// Wrap it over in case we come to the end of the array.
FOR i := nSlaveIndex+1 TO 9 DO
	IF i >= 9 THEN
		i := 1;
	END_IF
	IF cfg.aDevUsed[i] THEN
		M_GetNextSlaveIndex	:= i;
		RETURN;
	END_IF
END_FOR
END_METHOD

METHOD M_SetCommand : BOOL
VAR_IN_OUT
	nSlaveIndex:	INT;
	nAddressIndex:	INT;	// Which address space to read
END_VAR
VAR
	nNextSlaveIndex:		INT;
END_VAR
// We always read from JUMO
ctrl.nCmdType	:= E_MODBUS_CMD_TYPE.READ;

// Go to next register address to read
nAddressIndex	:= nAddressIndex + 1;
ctrl.nSlaveID	:= cfg.aSlaveID[nSlaveIndex];

IF nAddressIndex = E_JUMO_ADDRESS.COMMON THEN
	ctrl.nRegister	:= cfg.nAddrCommon;
	ctrl.nWords		:= cfg.nWordsCommon;
	M_SetCommand	:= TRUE;
ELSIF nAddressIndex = E_JUMO_ADDRESS.SET_POINTS THEN
	ctrl.nRegister	:= cfg.nAddrSetPoints;
	ctrl.nWords		:= cfg.nWordsSetPoints;
	M_SetCommand	:= TRUE;
ELSIF nAddressIndex = E_JUMO_ADDRESS.END THEN
	// Start reading from common
	nAddressIndex 	:= E_JUMO_ADDRESS.COMMON;
	ctrl.nRegister	:= cfg.nAddrCommon;
	ctrl.nWords		:= cfg.nWordsCommon;
	// Go to next slave
	nNextSlaveIndex	:= M_GetNextSlaveIndex(nSlaveIndex);
	IF nNextSlaveIndex <= nSlaveIndex THEN
		// We completed a full read of all slaves. Restart from the first one.
		M_SetCommand	:= FALSE;
	ELSE
		M_SetCommand	:= TRUE;
	END_IF
	nSlaveIndex		:= nNextSlaveIndex;
	ctrl.nSlaveID	:= cfg.aSlaveID[nSlaveIndex];
END_IF
END_METHOD

METHOD M_UserConfigure : BOOL
VAR_INPUT
END_VAR
// TODO USER
// Add here real configuration

// JUMO SlaveIDs are set as 1..8
// Set them to match real configuration
//cfg.aSlaveID[1]	:= 1;
//cfg.aSlaveID[2]	:= 2;

// FB_JUMO can read 8 JUMO devices.
// By default only the first one is enabled.
// Here we enable first two (one TeePee unit).
//cfg.aDevUsed[1]	:= TRUE;
//cfg.aDevUsed[2]	:= TRUE;
END_METHOD

END_FUNCTION_BLOCK

// POUs/Devices/FB_LAKESHORE_RS
FUNCTION_BLOCK FB_LAKESHORE_RS EXTENDS FB_LAKESHORE_BASE
VAR_INPUT
END_VAR
VAR_OUTPUT
END_VAR
VAR

	{attribute 'OPC.UA.DA' := '0'}
	comm:		FB_RS_COMM_LAKESHORE;	// Instance of Lakeshore customized comm 
	
END_VAR

// Set references
//cfgRef	REF=cfg;
//ctrlRef	REF=ctrl;
//statRef	REF=stat;


(* Execute comm instance *)
comm(	in_bSimulation	:= in_bSimulation,
		in_nModel		:= in_nModel,
		in_sCmdSuffix	:= in_sCmdSuffix, 
		in_sReplySuffix	:= in_sReplySuffix, 
		in_nTimeout		:= 2000);


// Execute the base class object FB_RS_BASE
SUPER^();

METHOD M_Configure
VAR_INPUT
END_VAR
VAR
	cmdList_Init_218:	ARRAY [1..8] OF T_LAKESHORE_COMMAND := [
							(cmd := '*RST', 	nReplies := 0, 	nValues := 0,	offset := 0),
							(cmd := '*CLS', 	nReplies := 0, 	nValues := 0,	offset := 0),
							(cmd := '*IDN?', 	nReplies := 1, 	nValues := 1,	offset := 0),
							(cmd := 'MODE 1', 	nReplies := 0, 	nValues := 0,	offset := 0),
							(cmd := '', 		nReplies := 0, 	nValues := 0,	offset := 0),
							(cmd := '', 		nReplies := 0, 	nValues := 0,	offset := 0),
							(cmd := '', 		nReplies := 0, 	nValues := 0,	offset := 0),
							(cmd := '', 		nReplies := 0, 	nValues := 0,	offset := 0)];

	cmdList_Init_340:	ARRAY [1..8] OF T_LAKESHORE_COMMAND := [
							(cmd := '*RST', 	nReplies := 0, 	nValues := 0,	offset := 0),
							(cmd := '*CLS', 	nReplies := 0, 	nValues := 0,	offset := 0),
							(cmd := '*IDN?', 	nReplies := 1, 	nValues := 1,	offset := 0),
							(cmd := 'MODE 2', 	nReplies := 0, 	nValues := 0,	offset := 0),
							(cmd := '', 		nReplies := 0, 	nValues := 0,	offset := 0),
							(cmd := '', 		nReplies := 0, 	nValues := 0,	offset := 0),
							(cmd := '', 		nReplies := 0, 	nValues := 0,	offset := 0),
							(cmd := '', 		nReplies := 0, 	nValues := 0,	offset := 0)];


	(*	List of READ commands *)
	(* Lakeshore 218 commands:
		Command "KRDG? 0" requests all 8 temperature values in K.
		Command "CRDG? 0" requests all 8 temperature values in C.
		Reply format: 
			+nn.nnn,+nn.nnn,+nn.nnn,+nn.nnn,+nn.nnn,+nn.nnn,+nn.nnn,+nn.nnn<CR><LF>
	*)
	cmdList_Read_218:	ARRAY [1..16] OF T_LAKESHORE_COMMAND := [
							(cmd := 'KRDG? 0', 	nReplies := 1, 	nValues := 8,	offset := 0),
							(cmd := 'CRDG? 0', 	nReplies := 1, 	nValues := 8,	offset := 8),
							(cmd := '', 		nReplies := 0, 	nValues := 0,	offset := 0),
							(cmd := '', 		nReplies := 0, 	nValues := 0,	offset := 0),
							(cmd := '', 		nReplies := 0, 	nValues := 0,	offset := 0),
							(cmd := '', 		nReplies := 0, 	nValues := 0,	offset := 0),
							(cmd := '', 		nReplies := 0, 	nValues := 0,	offset := 0),
							(cmd := '', 		nReplies := 0, 	nValues := 0,	offset := 0),
							(cmd := '', 		nReplies := 0, 	nValues := 0,	offset := 0),
							(cmd := '', 		nReplies := 0, 	nValues := 0,	offset := 0),
							(cmd := '', 		nReplies := 0, 	nValues := 0,	offset := 0),
							(cmd := '', 		nReplies := 0, 	nValues := 0,	offset := 0),
							(cmd := '', 		nReplies := 0, 	nValues := 0,	offset := 0),
							(cmd := '', 		nReplies := 0, 	nValues := 0,	offset := 0),
							(cmd := '', 		nReplies := 0, 	nValues := 0,	offset := 0),
							(cmd := '', 		nReplies := 0, 	nValues := 0,	offset := 0)];

	cmdList_Read_340:	ARRAY [1..16] OF T_LAKESHORE_COMMAND := [
							(cmd := 'KRDG? A', 	nReplies := 1, 	nValues := 1,	offset := 0),
							(cmd := 'KRDG? B', 	nReplies := 1, 	nValues := 1,	offset := 1),
							(cmd := 'SETP? 1', 	nReplies := 1, 	nValues := 1,	offset := 2),
							(cmd := 'PID? 1', 	nReplies := 1, 	nValues := 3,	offset := 3),
							(cmd := 'RAMP? 1', 	nReplies := 1, 	nValues := 2,	offset := 6),
							(cmd := 'RANGE?', 	nReplies := 1, 	nValues := 1,	offset := 8),
							(cmd := 'HTR?', 	nReplies := 1, 	nValues := 1,	offset := 9),
							(cmd := 'AOUT? 1', 	nReplies := 1, 	nValues := 1,	offset := 10),
							(cmd := 'AOUT? 2', 	nReplies := 1, 	nValues := 1,	offset := 11),
							(cmd := 'SETP? 2', 	nReplies := 1, 	nValues := 1,	offset := 12),
							(cmd := 'PID? 2', 	nReplies := 1, 	nValues := 3,	offset := 13),
							(cmd := '', 		nReplies := 0, 	nValues := 0,	offset := 0),
							(cmd := '', 		nReplies := 0, 	nValues := 0,	offset := 0),
							(cmd := '', 		nReplies := 0, 	nValues := 0,	offset := 0),
							(cmd := '', 		nReplies := 0, 	nValues := 0,	offset := 0),
							(cmd := '', 		nReplies := 0, 	nValues := 0,	offset := 0)];

	
END_VAR
// Execute base FB M_Configure().
// This will set cfg.nModel
SUPER^.M_Configure();

// TODO
// Populate cfg.cmdList_Init and cmdList_Read tables for the specific cfg.nModel.
IF cfg.nModel = 218 THEN
	cfg.cmdList_Init	:= cmdList_Init_218;
	cfg.cmdList_Read	:= cmdList_Read_218;
ELSIF cfg.nModel = 340 THEN
	cfg.cmdList_Init	:= cmdList_Init_340;
	cfg.cmdList_Read	:= cmdList_Read_340;
END_IF


// Set pointers to comm, i.e.
ptrCommCfg	:= ADR(comm.cfg);	(* Pointer to comm.cfg instance *)
ptrCommCtrl	:= ADR(comm.ctrl);	(* Pointer to comm.ctrl instance *)
ptrCommStat	:= ADR(comm.stat);	(* Pointer to comm.stat instance *)

// Set comm suffixes for commands and replies
ptrCommCfg^.sCmdSuffix		:= in_sCmdSuffix;
ptrCommCfg^.sReplySuffix	:= in_sReplySuffix;
END_METHOD

METHOD M_GetCommInitialised : BOOL
VAR_INPUT
END_VAR
// TODO: In each extended FB add the following:
// M_GetCommInitialised	:= comm.M_GetInitialised();

// This is just a dummy method for BASE FB
M_GetCommInitialised	:= comm.M_GetInitialised();
END_METHOD

METHOD M_GetCommStatus : E_RS_COMM_STATUS
VAR_INPUT
END_VAR
M_GetCommStatus	:= comm.M_GetStatus();
END_METHOD

METHOD M_GetCouplerState : BOOL
VAR_INPUT
END_VAR
IF comm.i_nCouplerState = 8  OR  in_bSimulation  THEN
	M_GetCouplerState	:= TRUE;	
ELSE
	M_GetCouplerState	:= FALSE;	
END_IF
END_METHOD

METHOD M_UpdateStatus
VAR_INPUT
END_VAR
// TODO
//
// Copy values from stat.lrReadings to correspondig stat variables.
// Check M_Configure(). It has to match!
//
// This is an example for model 340.
// This method has to match the list of commands in T_LAKESHORE_CFG::cmdList_Read
IF cfg.nModel = 218 THEN
	// Nothing to do.
	// NOTE: 8 readings [K]: stat.lrArrReadings[0..7]
	// NOTE: 8 readings [C]: stat.lrArrReadings[8..15]
	;	
ELSIF cfg.nModel = 340 THEN
	stat.lrKRDG_A	:= stat.lrArrReadings[0].lrValue;
	stat.lrCRDG_A	:= stat.lrKRDG_A - 273.15;
	stat.lrKRDG_B	:= stat.lrArrReadings[1].lrValue;
	stat.lrCRDG_B	:= stat.lrKRDG_B - 273.15;
	stat.lrSETP		:= stat.lrArrReadings[2].lrValue;
	stat.nPID_P		:= LREAL_TO_UINT(stat.lrArrReadings[3].lrValue);
	stat.nPID_I		:= LREAL_TO_UINT(stat.lrArrReadings[4].lrValue);
	stat.nPID_D		:= LREAL_TO_UINT(stat.lrArrReadings[5].lrValue);
	stat.bRAMP_On	:= LREAL_TO_BOOL(stat.lrArrReadings[6].lrValue);
	stat.lrRAMP_Rate:= stat.lrArrReadings[7].lrValue;
	stat.nRANGE		:= LREAL_TO_UINT(stat.lrArrReadings[8].lrValue);
	stat.lrHTR		:= stat.lrArrReadings[9].lrValue;
	stat.lrAOUT1	:= stat.lrArrReadings[10].lrValue;
	stat.lrAOUT2	:= stat.lrArrReadings[11].lrValue;
	stat.lrSETP2	:= stat.lrArrReadings[12].lrValue;
	stat.nPID2_P	:= LREAL_TO_UINT(stat.lrArrReadings[13].lrValue);
	stat.nPID2_I	:= LREAL_TO_UINT(stat.lrArrReadings[14].lrValue);
	stat.nPID2_D	:= LREAL_TO_UINT(stat.lrArrReadings[15].lrValue);
END_IF
END_METHOD

END_FUNCTION_BLOCK

// VISUs/Templates/GUI_TEMPLATE_CCC
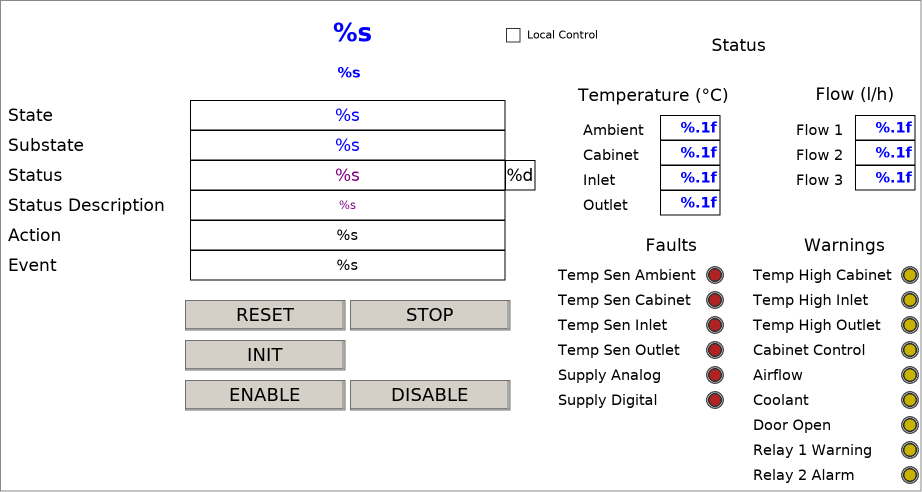
VISUALIZATION GUI_TEMPLATE_CCC  // 922x492
VAR_IN_OUT
	m_Instance:	FB_CCC;
END_VAR
    Rectangle (190,100 315x30), "%s", text variable: m_Instance.stat.sState
    Rectangle (190,130 315x30), "%s", text variable: m_Instance.stat.sSubstate
    Button (185,300 160x30), "RESET", input disabled if: (m_Instance.stat.bLocal = FALSE) <> 0
        OnMouseClick: execute { m_Instance.ctrl.nCommand := E_RS_COMMAND.RESET; m_Instance.ctrl.bExecute := TRUE; }
    Button (185,340 160x30), "INIT", input disabled if: (m_Instance.stat.bLocal = FALSE) <> 0
        OnMouseClick: execute { m_Instance.ctrl.nCommand := E_RS_COMMAND.INIT; m_Instance.ctrl.bExecute := TRUE; }
    Button (350,300 160x30), "STOP", input disabled if: (m_Instance.stat.bLocal = FALSE) <> 0
        OnMouseClick: execute { m_Instance.ctrl.nCommand := E_RS_COMMAND.STOP; m_Instance.ctrl.bExecute := TRUE; }
    Button (185,380 160x30), "ENABLE", input disabled if: (m_Instance.stat.bLocal = FALSE) <> 0
        OnMouseClick: execute { m_Instance.ctrl.nCommand := E_RS_COMMAND.ENABLE; m_Instance.ctrl.bExecute := TRUE; }
    Button (350,380 160x30), "DISABLE", input disabled if: (m_Instance.stat.bLocal = FALSE) <> 0
        OnMouseClick: execute { m_Instance.ctrl.nCommand := E_RS_COMMAND.DISABLE; m_Instance.ctrl.bExecute := TRUE; }
    Rectangle (5,100 180x30), "State"
    Rectangle (5,130 180x30), "Substate"
    Rectangle (190,160 315x30), "%s", text variable: m_Instance.stat.sStatus
    Rectangle (190,190 315x30), "%s", text variable: m_Instance.stat.sErrorText
    Rectangle (5,160 180x30), "Status"
    Rectangle (5,190 180x30), "Status Description"
    Rectangle (190,220 315x30), "%s", text variable: m_Instance.stat.sActionDesc
    Rectangle (190,250 315x30), "%s", text variable: m_Instance.stat.sEventDesc
    Rectangle (5,220 180x30), "Action"
    Rectangle (5,250 180x30), "Event"
    Rectangle (266,15 173x35), "%s", text variable: m_Instance.in_sName
    Checkbox (504,20 116x30), "Local Control", variable: m_Instance.stat.bLocal
    Rectangle (693,30 92x30), "Status"
    Rectangle (505,160 30x30), "%d", text variable: m_Instance.stat.nStatus
    Rectangle (569,80 169x30), "Temperature (°C)"
    Rectangle (806,79 98x30), "Flow (l/h)"
    Rectangle (580,115 70x30), "Ambient"
    Rectangle (580,140 70x30), "Cabinet"
    Rectangle (580,165 70x30), "Inlet"
    Rectangle (580,190 70x30), "Outlet"
    Rectangle (660,115 60x25), "%.1f", text variable: m_Instance.stat.lrTemp_ambient
    Rectangle (660,140 60x25), "%.1f", text variable: m_Instance.stat.lrTemp_cabinet
    Rectangle (660,165 60x25), "%.1f", text variable: m_Instance.stat.lrTemp_inlet
    Rectangle (660,190 60x25), "%.1f", text variable: m_Instance.stat.lrTemp_outlet
    Rectangle (855,115 60x25), "%.1f", text variable: m_Instance.stat.lrFlow_1
    Rectangle (781,115 65x30), "Flow 1"
    Rectangle (781,140 65x30), "Flow 2"
    Rectangle (855,140 60x25), "%.1f", text variable: m_Instance.stat.lrFlow_2
    Rectangle (781,165 65x30), "Flow 3"
    Rectangle (855,165 60x25), "%.1f", text variable: m_Instance.stat.lrFlow_3
    Rectangle (605,230 133x30), "Faults"
    Rectangle (555,260 150x30), "Temp Sen Ambient"
    Lamp1 (705,265 20x20), variable: m_Instance.stat.bFault_temp_sensor_ambient, style: Lamp-Lamp1-Red
    Rectangle (555,285 150x30), "Temp Sen Cabinet"
    Lamp1 (705,290 20x20), variable: m_Instance.stat.bFault_temp_sensor_cabinet, style: Lamp-Lamp1-Red
    Rectangle (555,310 150x30), "Temp Sen Inlet"
    Lamp1 (705,315 20x20), variable: m_Instance.stat.bFault_temp_sensor_inlet, style: Lamp-Lamp1-Red
    Rectangle (555,335 150x30), "Temp Sen Outlet"
    Lamp1 (705,340 20x20), variable: m_Instance.stat.bFault_temp_sensor_outlet, style: Lamp-Lamp1-Red
    Rectangle (555,360 150x30), "Supply Analog"
    Lamp1 (705,365 20x20), variable: m_Instance.stat.bFault_analog_supply, style: Lamp-Lamp1-Red
    Rectangle (555,385 150x30), "Supply Digital"
    Lamp1 (705,390 20x20), variable: m_Instance.stat.bFault_digital_supply, style: Lamp-Lamp1-Red
    Rectangle (778,230 133x30), "Warnings"
    Rectangle (750,260 150x30), "Temp High Cabinet"
    Lamp1 (900,265 20x20), variable: m_Instance.stat.bWarn_cabinet_high, style: Lamp-Lamp1-Yellow
    Rectangle (750,335 150x30), "Cabinet Control"
    Lamp1 (900,340 20x20), variable: m_Instance.stat.bWarn_cabinet_no_control, style: Lamp-Lamp1-Yellow
    Rectangle (750,310 150x30), "Temp High Outlet"
    Lamp1 (900,315 20x20), variable: m_Instance.stat.bWarn_outlet_high, style: Lamp-Lamp1-Yellow
    Rectangle (750,285 150x30), "Temp High Inlet"
    Lamp1 (900,290 20x20), variable: m_Instance.stat.bWarn_inlet_high, style: Lamp-Lamp1-Yellow
    Rectangle (750,360 150x30), "Airflow"
    Lamp1 (900,365 20x20), variable: m_Instance.stat.bWarn_airflow_insufficient, style: Lamp-Lamp1-Yellow
    Rectangle (750,385 150x30), "Coolant"
    Lamp1 (900,390 20x20), variable: m_Instance.stat.bWarn_coolant_insufficient, style: Lamp-Lamp1-Yellow
    Rectangle (750,410 150x30), "Door Open"
    Lamp1 (900,415 20x20), variable: m_Instance.stat.bWarn_door_open, style: Lamp-Lamp1-Yellow
    Rectangle (750,435 150x30), "Relay 1 Warning"
    Lamp1 (900,440 20x20), variable: m_Instance.stat.bWarn_relay1_warning, style: Lamp-Lamp1-Yellow
    Rectangle (750,460 150x30), "Relay 2 Alarm"
    Lamp1 (900,465 20x20), variable: m_Instance.stat.bWarn_relay2_alarm, style: Lamp-Lamp1-Yellow
    Rectangle (184,60 330x25), "%s", text variable: m_Instance.stat.sDeviceID
END_VISUALIZATION

// VISUs/Templates/GUI_TEMPLATE_LAKESHORE_340
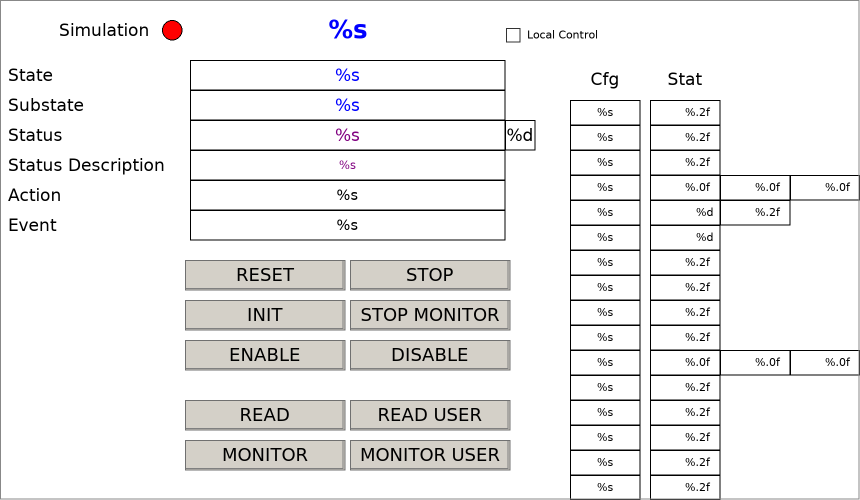
VISUALIZATION GUI_TEMPLATE_LAKESHORE_340  // 860x500
VAR_IN_OUT
	m_Instance:	FB_LAKESHORE_RS;
END_VAR
    Rectangle (190,60 315x30), "%s", text variable: m_Instance.stat.sState
    Rectangle (190,90 315x30), "%s", text variable: m_Instance.stat.sSubstate
    Button (185,260 160x30), "RESET", input disabled if: (m_Instance.stat.bLocal = FALSE) <> 0
        OnMouseClick: execute { m_Instance.ctrl.nCommand := E_RS_COMMAND.RESET; m_Instance.ctrl.bExecute := TRUE; }
    Button (185,300 160x30), "INIT", input disabled if: (m_Instance.stat.bLocal = FALSE) <> 0
        OnMouseClick: execute { m_Instance.ctrl.nCommand := E_RS_COMMAND.INIT; m_Instance.ctrl.bExecute := TRUE; }
    Button (350,260 160x30), "STOP", input disabled if: (m_Instance.stat.bLocal = FALSE) <> 0
        OnMouseClick: execute { m_Instance.ctrl.nCommand := E_RS_COMMAND.STOP; m_Instance.ctrl.bExecute := TRUE; }
    Button (185,340 160x30), "ENABLE", input disabled if: (m_Instance.stat.bLocal = FALSE) <> 0
        OnMouseClick: execute { m_Instance.ctrl.nCommand := E_RS_COMMAND.ENABLE; m_Instance.ctrl.bExecute := TRUE; }
    Button (350,340 160x30), "DISABLE", input disabled if: (m_Instance.stat.bLocal = FALSE) <> 0
        OnMouseClick: execute { m_Instance.ctrl.nCommand := E_RS_COMMAND.DISABLE; m_Instance.ctrl.bExecute := TRUE; }
    Rectangle (5,60 180x30), "State"
    Rectangle (5,90 180x30), "Substate"
    Rectangle (190,120 315x30), "%s", text variable: m_Instance.stat.sStatus
    Rectangle (190,150 315x30), "%s", text variable: m_Instance.stat.sErrorText
    Rectangle (5,120 180x30), "Status"
    Rectangle (5,150 180x30), "Status Description"
    Rectangle (190,180 315x30), "%s", text variable: m_Instance.stat.sActionDesc
    Rectangle (190,210 315x30), "%s", text variable: m_Instance.stat.sEventDesc
    Rectangle (5,180 180x30), "Action"
    Rectangle (5,210 180x30), "Event"
    Rectangle (232,12 232x35), "%s", text variable: m_Instance.in_sName
    Rectangle (574,64 62x30), "Cfg"
    Checkbox (504,20 116x30), "Local Control", variable: m_Instance.stat.bLocal
    Rectangle (505,120 30x30), "%d", text variable: m_Instance.stat.nStatus
    Button (185,400 160x30), "READ", tooltip "Single read of all commands in the configuration", input disabled if: (m_Instance.stat.bLocal = FALSE) <> 0
        OnMouseClick: execute { m_Instance.ctrl.nCommand := E_RS_COMMAND.READ; m_Instance.ctrl.bExecute := TRUE; }
    Button (350,400 160x30), "READ USER", tooltip "Single read of user command", input disabled if: (m_Instance.stat.bLocal = FALSE) <> 0
        OnMouseClick: execute { m_Instance.ctrl.nCommand := E_RS_COMMAND.READ_USER; m_Instance.ctrl.bExecute := TRUE; }
    Button (185,440 160x30), "MONITOR", tooltip "Continuously read all commands in the configuration", input disabled if: (m_Instance.stat.bLocal = FALSE) <> 0
        OnMouseClick: execute { m_Instance.ctrl.nCommand := E_RS_COMMAND.MONITOR; m_Instance.ctrl.bExecute := TRUE; }
    Button (350,440 160x30), "MONITOR USER", tooltip "Continuously read the User command", input disabled if: (m_Instance.stat.bLocal = FALSE) <> 0
        OnMouseClick: execute { m_Instance.ctrl.nCommand := E_RS_COMMAND.MONITOR_USER; m_Instance.ctrl.bExecute := TRUE; }
    Rectangle (570,100 70x25), "%s", text variable: m_Instance.cfg.cmdList_Read[1].cmd
    Rectangle (570,125 70x25), "%s", text variable: m_Instance.cfg.cmdList_Read[2].cmd
    Rectangle (570,150 70x25), "%s", text variable: m_Instance.cfg.cmdList_Read[3].cmd
    Rectangle (570,175 70x25), "%s", text variable: m_Instance.cfg.cmdList_Read[4].cmd
    Rectangle (570,200 70x25), "%s", text variable: m_Instance.cfg.cmdList_Read[5].cmd
    Rectangle (570,225 70x25), "%s", text variable: m_Instance.cfg.cmdList_Read[6].cmd
    Rectangle (570,250 70x25), "%s", text variable: m_Instance.cfg.cmdList_Read[7].cmd
    Rectangle (570,275 70x25), "%s", text variable: m_Instance.cfg.cmdList_Read[8].cmd
    Rectangle (570,300 70x25), "%s", text variable: m_Instance.cfg.cmdList_Read[9].cmd
    Rectangle (570,325 70x25), "%s", text variable: m_Instance.cfg.cmdList_Read[10].cmd
    Rectangle (570,350 70x25), "%s", text variable: m_Instance.cfg.cmdList_Read[11].cmd
    Rectangle (570,375 70x25), "%s", text variable: m_Instance.cfg.cmdList_Read[12].cmd
    Rectangle (570,400 70x25), "%s", text variable: m_Instance.cfg.cmdList_Read[13].cmd
    Rectangle (570,425 70x25), "%s", text variable: m_Instance.cfg.cmdList_Read[14].cmd
    Rectangle (570,450 70x25), "%s", text variable: m_Instance.cfg.cmdList_Read[15].cmd
    Rectangle (570,475 70x25), "%s", text variable: m_Instance.cfg.cmdList_Read[16].cmd
    Rectangle (650,100 70x25), "%.2f", text variable: m_Instance.stat.lrArrReadings[0].lrValue
    Rectangle (650,125 70x25), "%.2f", text variable: m_Instance.stat.lrArrReadings[1].lrValue
    Rectangle (650,150 70x25), "%.2f", text variable: m_Instance.stat.lrArrReadings[2].lrValue
    Rectangle (650,175 70x25), "%.0f", text variable: m_Instance.stat.lrArrReadings[3].lrValue
    Rectangle (720,175 70x25), "%.0f", text variable: m_Instance.stat.lrArrReadings[4].lrValue
    Rectangle (790,175 70x25), "%.0f", text variable: m_Instance.stat.lrArrReadings[5].lrValue
    Rectangle (650,200 70x25), "%d", text variable: m_Instance.stat.bRAMP_On
    Rectangle (720,200 70x25), "%.2f", text variable: m_Instance.stat.lrRAMP_Rate
    Rectangle (650,250 70x25), "%.2f", text variable: m_Instance.stat.lrArrReadings[9].lrValue
    Rectangle (650,275 70x25), "%.2f", text variable: m_Instance.stat.lrArrReadings[10].lrValue
    Rectangle (720,350 70x25), "%.0f", text variable: m_Instance.stat.lrArrReadings[14].lrValue
    Rectangle (790,350 70x25), "%.0f", text variable: m_Instance.stat.lrArrReadings[15].lrValue
    Rectangle (650,300 70x25), "%.2f", text variable: m_Instance.stat.lrArrReadings[11].lrValue
    Rectangle (650,325 70x25), "%.2f", text variable: m_Instance.stat.lrArrReadings[12].lrValue
    Rectangle (650,350 70x25), "%.0f", text variable: m_Instance.stat.lrArrReadings[13].lrValue
    Rectangle (650,375 70x25), "%.2f", text variable: m_Instance.stat.lrArrReadings[16].lrValue
    Rectangle (650,400 70x25), "%.2f", text variable: m_Instance.stat.lrArrReadings[17].lrValue
    Rectangle (650,425 70x25), "%.2f", text variable: m_Instance.stat.lrArrReadings[18].lrValue
    Rectangle (650,450 70x25), "%.2f", text variable: m_Instance.stat.lrArrReadings[19].lrValue
    Rectangle (650,475 70x25), "%.2f", text variable: m_Instance.stat.lrArrReadings[20].lrValue
    Rectangle (654,64 62x30), "Stat"
    Button (350,300 160x30), "STOP MONITOR", tooltip "Stop Monitoring if in OP/MONITORIN state.", input disabled if: (m_Instance.stat.bLocal = FALSE) <> 0
        OnMouseClick: execute { m_Instance.ctrl.nCommand := E_RS_COMMAND.STOPMON; m_Instance.ctrl.bExecute := TRUE; }
    Rectangle (650,225 70x25), "%d", text variable: m_Instance.stat.lrArrReadings[8].lrValue
    Rectangle (56,15 101x30), "Simulation", invisible if: (m_Instance.stat.bSimulation=FALSE)
    Ellipse (162,20 20x20), tooltip "GREEN=Initialized RED=Not-initialized", text variable: m_Instance.stat.bInitialised, invisible if: (m_Instance.stat.bSimulation=FALSE)
END_VISUALIZATION

